		(*-----------------------Weiterschaltbedingungen----------------------------*)
		IF gb_memEndOfBandMarkNIO THEN
			fb_state_entry.i16_next_step := 370;
		ELSE
			IF gst_datensatz.st_md.b_tagreader_fahrend THEN
				(* Pille sofort beschreiben *)
				fb_state_entry.i16_next_step := 350;
			ELSE
				IF st_drive_cmd.enu_cmd = NO_COMMAND THEN
					(* Warte mit Pille beschreiben, bis der Bestücktisch im Ziel ist *)
					fb_state_entry.i16_next_step := 350;
				END_IF
			END_IF
		END_IF


		IF	gst_datensatz.st_md.b_wt_transport_aktiv =FALSE THEN
			visu.b_merker_vollbestuecken:= FALSE;
			s_alte_artikelnummer := '';
			fb_state_entry.i16_next_step := 360;
		END_IF

		IF fb_state_entry.X THEN
			Teile_nach_Bandwechsel:= FALSE;
			IF gst_datensatz.st_wkz.i16_anzahl_Teile_autostop_bandwechsel <> 0 THEN
				gi16_anzahl_Teile_autostop_bandwechsel := gi16_anzahl_Teile_autostop_bandwechsel + 1;
			END_IF
		END_IF

(*=======================================================*)
	350: (* Schreibe Daten auf Tag *)
		IF fb_state_entry.E THEN
			(* Auswertung der Bestückung (Pins bzw. Rasterplatte) des ISK *)
			ST_Markiere_WT_IO();
		END_IF

		(*-----------------------Weiterschaltbedingungen----------------------------*)
		IF balluff_tag_reader.st_ctrl.out.b_fertig AND NOT fb_state_entry.E THEN
			balluff_tag_reader.st_ctrl.in.b_start_schreiben := FALSE;
			fb_state_entry.i16_next_step := 360;
		END_IF

(*=======================================================*)
	360:	(* Aktualisiere letztes benutzes Werkzeug *)
		IF fb_state_entry.E THEN
			ST_Schreibe_LastUsedTool();
		END_IF

		(*-----------------------Weiterschaltbedingungen----------------------------*)
		IF balluff_tag_reader.st_ctrl.out.b_fertig AND NOT fb_state_entry.E THEN
			balluff_tag_reader.st_ctrl.in.b_start_schreiben := FALSE;
			IF gst_datensatz.st_md.b_tagreader_fahrend THEN
				fb_state_entry.i16_next_step := 370;
			ELSE
				fb_state_entry.i16_next_step := 380;
				fb_Z_Achse_ausfahren(b_start:= FALSE, t_zeit=>t_Z_Achse_ausfahren );
			END_IF
		END_IF

(*=======================================================*)
	370:	(* Warte noch auf die Z-Achse, bis sie auf der Übergabeposition steht. *)

		gb_memEndOfBandMarkNIO := FALSE;

		(*-----------------------Weiterschaltbedingungen----------------------------*)
		IF st_drive_cmd.enu_cmd = NO_COMMAND THEN
			fb_state_entry.i16_next_step := 380;
			fb_Z_Achse_ausfahren(b_start:= FALSE, t_zeit=>t_Z_Achse_ausfahren );
		END_IF

(*=======================================================*)
	380:

		CASE gst_datensatz.st_md.i16_typ_zelle OF
			KEINE_ZELLE:
				;

			BESTUECKZELLE_1700:
				(*-----------------------Weiterschaltbedingungen----------------------------*)
				fb_state_entry.i16_next_step := BEREIT;

			RASTERFOLIE:
				(*-----------------------Weiterschaltbedingungen----------------------------*)
				IF rasterfolienmontage.st_ctrl.out.b_fertig_2 THEN
					fb_state_entry.i16_next_step := BEREIT;
				END_IF
		END_CASE

		IF fb_state_entry.X THEN
			(* Stoppe Bestückzeit *)
			zeit_wt_bestuecken := TIME_TO_DWORD(fb_ton_taktzeitmessung_bestuecken.ET);
			fb_ton_taktzeitmessung_bestuecken.IN := FALSE;
			(* Starte WT Wechselzeit *)
			fb_ton_taktzeitmessung_wt_wechsel.IN := TRUE;
		END_IF

(*==========================Bestückzelle1720=============================*)
	395: (*Warten bis keine ander Produktions Meldung ansteht *)
		IF	TestAndSet(ST_Message_Produktion.LockFlag) THEN
			ST_Message_Produktion.ClearMessageLines();
			fb_state_entry.i16_next_step := 396;
		END_IF

(*=======================================================*)
	396:  (*Produktions Meldung*)
		Visu.MeldungProduktion.Color_R := 255;
		Visu.MeldungProduktion.Color_G := 0;
		Visu.MeldungProduktion.Color_B := 0;
		IF visu.s_akt_sprache = 'de' THEN
			Visu.MeldungProduktion.Name:='Zelle war nicht in Betrieb, bitte Instandhalter informieren!$R$N$R$NÖler,Bestückposition, Seitenversatz und Biegewinkel kontrollieren$R$NMeldung kann nur eingeloggt quittiert werden';
		ELSIF visu.s_akt_sprache = 'en' THEN
			Visu.MeldungProduktion.Name:='Station has not been used for last order, please inform Maintenance Technician!$R$N$R$Ncheck oiler, stich position, left/right and bending angle$R$Nmessage can only be acknowledged when logged in';
		ELSIF visu.s_akt_sprache = 'cz' THEN
			Visu.MeldungProduktion.Name:='Bunka nebyla v provozu, informujte prosim serizovace. Zkontrolujte olej, nastaveni os a uhel ohybu.$R$NZprávu lze potvrdit jen po prihlaseni ';
		END_IF
		Visu.MeldungProduktion.ShowMessage := TRUE;
		Visu.MeldungProduktion.Button1.sichtbar:=TRUE;	(*OK*)
		Visu.MeldungProduktion.Button1.Text:='Ok';

		(*-----------------------Weiterschaltbedingungen----------------------------*)
		IF visu.b_logon THEN
			IF Visu.MeldungProduktion.Button1.tasten THEN
				IF gst_datensatz.st_md.	b_tagreader_fahrend THEN
					fb_state_entry.i16_next_step := 400;
				ELSE
					fb_state_entry.i16_next_step := 405;
				END_IF
			END_IF
		END_IF

		IF fb_state_entry.X THEN
			gst_PersDaten.b_Zelle_nicht_in_Betrieb := FALSE;
		END_IF

(*=======================================================*)
	400:	(* Fahre Z-Achse bis auf die erste Bestückposition *)
		IF fb_state_entry.E THEN
			(* Z-Achse verfahren *)
			fb_axis.lr_soll_geschwindigkeit := gst_datensatz.st_wkz.r_auto_z;
			fb_axis.st_position.r_soll := gst_datensatz.st_isk.lr_pos_z_0 + gst_datensatz.st_wkz.lr_offset_z_pos_0 + gst_datensatz.st_wt.lr_offset_z_pos_0 + gst_datensatz.st_md.lr_offset_z_pos_0 + gst_datensatz.st_bestueckprogramm.lr_z[0];
			st_drive_cmd.enu_cmd := MOVE_ABSOLUTE;
		END_IF

		(*-----------------------Weiterschaltbedingungen----------------------------*)
		(* Z-Achse losfahren und währenddessen beschreibt der Tagreader die Pille *)
		fb_state_entry.i16_next_step := 405;

(*=======================================================*)
	405:	(*  WT als schlecht markieren*)
		IF fb_state_entry.E THEN
			ST_Markiere_WT_NIO();
		END_IF

		(*-----------------------Weiterschaltbedingungen----------------------------*)
		IF balluff_tag_reader.st_ctrl.out.b_fertig AND NOT fb_state_entry.E THEN
			(* Ok: Daten sind auf der Pille *)
			balluff_tag_reader.st_ctrl.in.b_start_schreiben := FALSE;
			IF gst_datensatz.st_md.b_tagreader_fahrend THEN
				(* Warte auf Z-Achse *)
				fb_state_entry.i16_next_step := 410;
			ELSE
				(* Daten geschrieben und erst jetzt die Z-Achse fahren *)
				fb_state_entry.i16_next_step := 420;
			END_IF
		END_IF

(*=======================================================*)
	410:	(* Warte noch auf die Z-Achse, bis sie im Ziel steht. *)

		(*-----------------------Weiterschaltbedingungen----------------------------*)
		IF st_drive_cmd.enu_cmd = NO_COMMAND THEN
			fb_state_entry.i16_next_step := 430;
		END_IF

(*=======================================================*)
	420:	(* Fahre Z-Achse bis auf die erste Bestückposition *)
		IF fb_state_entry.E THEN
			(* Z-Achse verfahren *)
			fb_axis.lr_soll_geschwindigkeit := gst_datensatz.st_wkz.r_auto_z;
			fb_axis.st_position.r_soll := gst_datensatz.st_isk.lr_pos_z_0 + gst_datensatz.st_wkz.lr_offset_z_pos_0 + gst_datensatz.st_wt.lr_offset_z_pos_0 + gst_datensatz.st_md.lr_offset_z_pos_0 + gst_datensatz.st_bestueckprogramm.lr_z[0];
			st_drive_cmd.enu_cmd := MOVE_ABSOLUTE;
		END_IF

		(*-----------------------Weiterschaltbedingungen----------------------------*)
		IF st_drive_cmd.enu_cmd = NO_COMMAND THEN
			fb_state_entry.i16_next_step := 430;
		END_IF

(*=======================================================*)
	430:	(* Führung wird an die Bestückachse abgegeben und die Z-Achse wird ausschliesslich über Kurvenscheiben-Kopplung verfahren *)
		IF fb_state_entry.E THEN
			fb_Z_Achse_einfahren(b_start:= FALSE, t_zeit=> t_Z_Achse_einfahren);
			fb_Bestueckung(b_start:= TRUE, t_zeit=> );
			axis_virt_master.st_ctrl.in.b_start := TRUE;

			(* Stoppe WT Wechselzeit *)
			zeit_wt_wechsel := TIME_TO_DWORD(fb_ton_taktzeitmessung_wt_wechsel.ET);
			fb_ton_taktzeitmessung_wt_wechsel.IN := FALSE;

			(* Starte Bestückzeit *)
			fb_ton_taktzeitmessung_bestuecken.IN := TRUE;
		END_IF

		(*-----------------------Weiterschaltbedingungen----------------------------*)
		IF NOT axis_virt_master.st_ctrl.out.b_fertig THEN
			axis_virt_master.st_ctrl.in.b_start := FALSE;
			fb_state_entry.i16_next_step := 440;
		END_IF

		IF fb_state_entry.X THEN
			(* Stoppe Bestückzeit *)
			zeit_wt_bestuecken := TIME_TO_DWORD(fb_ton_taktzeitmessung_bestuecken.ET);
			fb_ton_taktzeitmessung_bestuecken.IN := FALSE;

			(* Starte WT Wechselzeit *)
			fb_ton_taktzeitmessung_wt_wechsel.IN := TRUE;
		END_IF

(*=======================================================*)
	440:	(* Warte auf  Bestückachse fertig mit Pins setzen *)

		(*-----------------------Weiterschaltbedingungen----------------------------*)
		IF axis_virt_master.st_ctrl.out.b_fertig THEN
			fb_state_entry.i16_next_step := 450;
			fb_Bestueckung(b_start:=FALSE, t_zeit=>t_Bestueckung);
			fb_Z_Achse_ausfahren(b_start:= TRUE, t_zeit=> );
		END_IF

(*=======================================================*)
	450: (* Fahre Z-Achse zurück zur Übergabeposition *)
		IF fb_state_entry.E THEN
			 fb_axis.st_position.r_soll := gst_datensatz.st_md.st_md_z_achse.lr_wt_uebergabepos;
			st_drive_cmd.enu_cmd := MOVE_ABSOLUTE;
		END_IF

		(*Nach einem Bandwechsel soll nach X-Teilen gestoppt werden.*)
		IF gst_datensatz.st_wkz.i16_anzahl_Teile_autostop_bandwechsel > 0 THEN
			IF gi16_anzahl_Teile_autostop_bandwechsel = gst_datensatz.st_wkz.i16_anzahl_Teile_autostop_bandwechsel THEN
				gb_nach_bawe_einzelfertigung := TRUE;
			END_IF
		END_IF

		(*-----------------------Weiterschaltbedingungen----------------------------*)
		IF gst_datensatz.st_md.b_tagreader_fahrend THEN
			(* Pille sofort beschreiben *)
			fb_state_entry.i16_next_step := 460;
		ELSE
			IF st_drive_cmd.enu_cmd = NO_COMMAND THEN
				(* Warte mit Pille beschreiben *)
				fb_state_entry.i16_next_step := 460;
			END_IF
		END_IF

		IF	gst_datensatz.st_md.b_wt_transport_aktiv =FALSE THEN
			visu.b_merker_vollbestuecken:= FALSE;
			s_alte_artikelnummer := '';
			fb_state_entry.i16_next_step := 480;
		END_IF

		IF fb_state_entry.X THEN
			IF gst_datensatz.st_wkz.i16_anzahl_Teile_autostop_bandwechsel <> 0 THEN
				gi16_anzahl_Teile_autostop_bandwechsel := gi16_anzahl_Teile_autostop_bandwechsel + 1;
			END_IF
		END_IF

(*=======================================================*)
	460: (* Schreibe Daten auf Tag *)
		IF fb_state_entry.E THEN
			(* WT Hat die Maschine auf regulärem Weg wieder verlassen *)
			ST_Markiere_WT_IO();
		END_IF

		(*-----------------------Weiterschaltbedingungen----------------------------*)
		IF balluff_tag_reader.st_ctrl.out.b_fertig AND NOT fb_state_entry.E THEN
			balluff_tag_reader.st_ctrl.in.b_start_schreiben := FALSE;
			fb_state_entry.i16_next_step := 470;
		END_IF

(*=======================================================*)
	470:	(* aktualisiere letztes benutzes Werkzeug *)
		IF fb_state_entry.E THEN
			ST_Schreibe_LastUsedTool();
		END_IF

		IF balluff_tag_reader.st_ctrl.out.b_fertig AND NOT fb_state_entry.E THEN
			balluff_tag_reader.st_ctrl.in.b_start_schreiben := FALSE;
			IF gst_datensatz.st_md.b_tagreader_fahrend THEN
				fb_state_entry.i16_next_step := 480;
			ELSE
				fb_Z_Achse_ausfahren(b_start:= FALSE, t_zeit=> );
				fb_state_entry.i16_next_step := BEREIT;
			END_IF
		END_IF

(*=======================================================*)
	480:	(* Z-Achse ist fertig positioniert *)

		(*-----------------------Weiterschaltbedingungen----------------------------*)
		IF st_drive_cmd.enu_cmd = NO_COMMAND THEN
			fb_Z_Achse_ausfahren(b_start:= FALSE, t_zeit=> );
			fb_state_entry.i16_next_step := BEREIT;
		END_IF

(*=======================================================*)
	FEHLER:
		IF fb_state_entry.E THEN
			st_ctrl_out.b_fehler := TRUE;
			fb_ton_quitt.IN := FALSE;
			st_ctrl_out.b_busy:=FALSE;
		END_IF

		(*-----------------------Weiterschaltbedingungen----------------------------*)
		IF st_ctrl_in.b_quitt AND NOT fb_state_entry.E THEN
			st_ctrl_out.b_fehler := FALSE;
			st_drive_cmd.enu_cmd := RESET;
			st_drive_cmd_y_achse.enu_cmd := RESET;
			fb_ton_quitt.IN := TRUE;
		END_IF

		IF st_ctrl_in.b_stop AND NOT z_achse.Status.HasBeenStopped THEN
			st_drive_cmd.enu_cmd := STOP_AXIS;
		END_IF

		IF st_ctrl_in.b_halt AND z_achse.Status.Moving THEN
			st_drive_cmd.enu_cmd := HALT_AXIS;
			st_geschwindigkeiten.lr_verzoegerung := lr_decceleration_nothalt;
		END_IF

		IF fb_ton_quitt.Q THEN
			fb_ton_quitt.IN := FALSE;
			fb_state_entry.i16_next_step := INIT;
		END_IF

(*=======================================================*)
	STOP:
		IF fb_state_entry.E THEN
			st_ctrl_out.b_busy:=FALSE;
			IF z_achse.NcToPlc.CoupleState = 0 THEN
				st_drive_cmd.enu_cmd := STOP_AXIS;
			END_IF
		END_IF

		(*-----------------------Weiterschaltbedingungen----------------------------*)
		IF st_drive_cmd.enu_cmd = NO_COMMAND AND z_achse.Status.NotMoving THEN
			fb_state_entry.i16_next_step := STILLSTAND;
		END_IF

(*=======================================================*)
	STILLSTAND:
		IF fb_state_entry.E THEN
			st_drive_cmd.enu_cmd := POWER_DISABLE;
			fb_ton_quitt.IN := FALSE;
		END_IF

		(*-----------------------Weiterschaltbedingungen----------------------------*)
		IF st_ctrl_in.b_quitt AND NOT fb_state_entry.E THEN
			fb_ton_quitt.IN := TRUE;
		END_IF

		IF fb_ton_quitt.Q THEN
			fb_ton_quitt.IN := FALSE;
			fb_state_entry.i16_next_step := INIT;
		END_IF

(*=======================================================*)
	HALT:
		IF fb_state_entry.E THEN
			IF z_achse.NcToPlc.CoupleState = 0 THEN
				st_drive_cmd.enu_cmd := HALT_AXIS;
				st_geschwindigkeiten.lr_verzoegerung := lr_decceleration_nothalt;
			END_IF
			fb_ton_quitt.IN := FALSE;
		END_IF

		(*-----------------------Weiterschaltbedingungen----------------------------*)
		IF st_ctrl_in.b_quitt AND NOT fb_state_entry.E THEN
			fb_ton_quitt.IN := TRUE;
		END_IF

		IF fb_ton_quitt.Q THEN
			fb_ton_quitt.IN := FALSE;
			fb_state_entry.i16_next_step := INIT;
		END_IF

(*=======================================================*)
	HANDRAD:	(* Überprüfe Nullpunktverschiebung des Absolutwertgebers auf Korrektheit *)
		IF fb_state_entry.E THEN
			st_ctrl_out.b_fehler := TRUE;
			fb_axis.i16_nc_parameter_nummer := AxisEncoderOffset;
			st_drive_cmd.enu_cmd := READ_NC_PARAMETER;
		END_IF

		(*-----------------------Weiterschaltbedingungen----------------------------*)
		IF st_drive_cmd.enu_cmd = NO_COMMAND THEN
			IF fb_axis.r_wert_nc_read_parameter = gst_datensatz.st_md.st_md_z_achse.lr_nullpunktverschiebung THEN
				fb_state_entry.i16_next_step := 2040;	(* Jogbetrieb *)
			ELSE
				fb_state_entry.i16_next_step := 2010;	(* Reglerfreigabe nehmen und Nullpunktverschiebung schreiben *)
			END_IF
		END_IF

(*=======================================================*)
	2010:	(* Reglerfreigabe wegnehmen , damit Nullpunktverschiebung geschrieben werden kannt*)
		IF fb_state_entry.E THEN
			st_drive_cmd.enu_cmd := POWER_DISABLE;
		END_IF

		(*-----------------------Weiterschaltbedingungen----------------------------*)
		IF st_drive_cmd.enu_cmd = NO_COMMAND THEN
			fb_state_entry.i16_next_step := 2020;
		END_IF

(*=======================================================*)
	2020:	(* Nullpunktverschiebung hat sich geändert, deshalb erst Null reinschreiben, um keinen Additionsfehler zu machen, *)
			(* weil der Wert der Verschiebung beim Neustart komplett auf die Achse geschrieben wird *)
		IF fb_state_entry.E THEN
			fb_axis.i16_nc_parameter_nummer := AxisEncoderOffset;
			fb_axis.r_wert_nc_write_parameter := 0.0;
			st_drive_cmd.enu_cmd := WRITE_NC_PARAMETER;
		END_IF

		(*-----------------------Weiterschaltbedingungen----------------------------*)
		IF st_drive_cmd.enu_cmd = NO_COMMAND THEN
			fb_state_entry.i16_next_step := 2030;
		END_IF

(*=======================================================*)
	2030:	(* Aktuelle Nullpunktverschiebung des Absolutwertgebers an die Achse senden *)
		IF fb_state_entry.E THEN
			fb_axis.i16_nc_parameter_nummer := AxisEncoderOffset;
			fb_axis.r_wert_nc_write_parameter := gst_datensatz.st_md.st_md_z_achse.lr_nullpunktverschiebung;
			st_drive_cmd.enu_cmd := WRITE_NC_PARAMETER;
		END_IF

		(*-----------------------Weiterschaltbedingungen----------------------------*)
		IF st_drive_cmd.enu_cmd = NO_COMMAND THEN
			fb_state_entry.i16_next_step := 2040;
		END_IF

(*=======================================================*)
	2040:	(* Jogbetrieb *)
		IF fb_state_entry.E THEN
			fb_axis.lr_soll_geschwindigkeit := st_geschwindigkeiten.lr_jog;
		END_IF

		IF ST_Euchner_Handbedienpult.i16_Handrad_delta > 0 THEN
			st_drive_cmd.enu_cmd := JOG_VORWAERTS;
		ELSIF ST_Euchner_Handbedienpult.i16_Handrad_delta < 0 THEN
			st_drive_cmd.enu_cmd := JOG_RUECKWAERTS;
		ELSE
			IF z_achse.Status.Moving THEN
				st_drive_cmd.enu_cmd := JOG_STOP;
			END_IF
		END_IF

		(*-----------------------Weiterschaltbedingungen----------------------------*)
		IF gi16_betriebsart <> HAND OR NOT b_hand_dialog_aktiv THEN
			fb_state_entry.i16_next_step := 2050;
		END_IF

(*=======================================================*)
	2050:
		IF fb_state_entry.E THEN
			st_drive_cmd.enu_cmd := ABORT;
		END_IF

		(*-----------------------Weiterschaltbedingungen----------------------------*)
		IF st_drive_cmd.enu_cmd = NO_COMMAND THEN
			fb_state_entry.i16_next_step := 2060;
		END_IF

(*=======================================================*)
	2060:	(* Reglerfreigabe wegnehmen *)
		IF fb_state_entry.E THEN
			st_drive_cmd.enu_cmd := POWER_DISABLE;
		END_IF

		(*-----------------------Weiterschaltbedingungen----------------------------*)
		IF st_drive_cmd.enu_cmd = NO_COMMAND THEN
			st_ctrl_out.b_fehler := FALSE;
			fb_state_entry.i16_next_step := INIT;
		END_IF

(*=======================================================*)
	NULLPUNKT_SETZEN:
		(* Aktuellen Jog beenden, sonst Probleme beim Softwareendschalter*)
		IF fb_state_entry.E THEN
			st_drive_cmd.enu_cmd := JOG_STOP;
		END_IF

		(*-----------------------Weiterschaltbedingungen----------------------------*)
		IF st_drive_cmd.enu_cmd = NO_COMMAND THEN
			fb_state_entry.i16_next_step := 2505;
		END_IF

(*=======================================================*)
	2505:
		(* 	Lese aktuelle Nullpunkt verschiebung von der Hardware. Der Benutze könnte einen falschen
			Wert eingetragen haben *)
		IF fb_state_entry.E THEN
			fb_axis.i16_nc_parameter_nummer := AxisEncoderOffset;
			st_drive_cmd.enu_cmd := READ_NC_PARAMETER;
		END_IF

		(*-----------------------Weiterschaltbedingungen----------------------------*)
		IF st_drive_cmd.enu_cmd = NO_COMMAND THEN
			gst_datensatz.st_md.st_md_z_achse.lr_nullpunktverschiebung := fb_axis.r_wert_nc_read_parameter;
			fb_state_entry.i16_next_step := 2510;
		END_IF

(*=======================================================*)
	2510:	(* Nullpunktverschiebung berechnen *)
		IF fb_state_entry.E THEN
			lr_pos_ohneverschiebung := axis_z_achse.st_visu.lr_position_ist - gst_datensatz.st_md.st_md_z_achse.lr_nullpunktverschiebung;

			gst_datensatz.st_md.st_md_z_achse.lr_nullpunktverschiebung := - lr_pos_ohneverschiebung;
		END_IF

		(*-----------------------Weiterschaltbedingungen----------------------------*)
		(* Aktiviere den Wert in die Hardware *)
		fb_state_entry.i16_next_step := HANDRAD;

(*=======================================================*)
	INBETRIEBNAHME:	(* Überprüfe Nullpunktverschiebung des Absolutwertgebers auf Korrektheit *)
		IF fb_state_entry.E THEN
			fb_axis.i16_nc_parameter_nummer := AxisEncoderOffset;
			st_drive_cmd.enu_cmd := READ_NC_PARAMETER;
		END_IF

		(*-----------------------Weiterschaltbedingungen----------------------------*)
		IF st_drive_cmd.enu_cmd = NO_COMMAND THEN
			IF fb_axis.r_wert_nc_read_parameter = gst_datensatz.st_md.st_md_z_achse.lr_nullpunktverschiebung THEN
				fb_state_entry.i16_next_step := 5100;	(* Reversiersequenz*)
			ELSE
				fb_state_entry.i16_next_step := 5010;	(* Reglerfreigabe nehmen und Nullpunktverschiebung schreiben *)
			END_IF
		END_IF

(*=======================================================*)
	5010:	(* Reglerfreigabe wegnehmen, damit Nullpunktverschiebung geschrieben werden kannt*)
		IF fb_state_entry.E THEN
			st_drive_cmd.enu_cmd := POWER_DISABLE;
		END_IF

		(*-----------------------Weiterschaltbedingungen----------------------------*)
		IF st_drive_cmd.enu_cmd = NO_COMMAND THEN
			fb_state_entry.i16_next_step := 5020;
		END_IF

(*=======================================================*)
	5020:	(* Nullpunktverschiebung hat sich geändert, deshalb erst Null reinschreiben, um keinen Additionsfehler zu machen, *)
			(* weil der Wert der Verschiebung beim Neustart komplett auf die Achse geschrieben wird *)
		IF fb_state_entry.E THEN
			fb_axis.i16_nc_parameter_nummer := AxisEncoderOffset;
			fb_axis.r_wert_nc_write_parameter := 0.0;
			st_drive_cmd.enu_cmd := WRITE_NC_PARAMETER;
		END_IF

		(*-----------------------Weiterschaltbedingungen----------------------------*)
		IF st_drive_cmd.enu_cmd = NO_COMMAND THEN
			fb_state_entry.i16_next_step := 5030;
		END_IF

(*=======================================================*)
	5030:	(* Aktuelle Nullpunktverschiebung des Absolutwertgebers an die Achse senden *)
		IF fb_state_entry.E THEN
			fb_axis.i16_nc_parameter_nummer := AxisEncoderOffset;
			fb_axis.r_wert_nc_write_parameter := gst_datensatz.st_md.st_md_z_achse.lr_nullpunktverschiebung;
			st_drive_cmd.enu_cmd := WRITE_NC_PARAMETER;
		END_IF

		(*-----------------------Weiterschaltbedingungen----------------------------*)
		IF st_drive_cmd.enu_cmd = NO_COMMAND THEN
			fb_state_entry.i16_next_step := 5100;
		END_IF

(*=======================================================*)
	5100:	(* Verfahren der Achse zwischen zwei Punkten zum Testen verschiedener Achsparameter *)
		IF fb_state_entry.E THEN
			fb_axis.lr_soll_geschwindigkeit := st_geschwindigkeiten.lr_jog;
			fb_axis.st_position.lr_ibn_pos_start := 10.0;
			fb_axis.st_position.lr_ibn_pos_ziel := -10.0;
		END_IF

		(*-----------------------Weiterschaltbedingungen----------------------------*)
		IF st_ctrl_in.b_ibn_start THEN
			fb_state_entry.i16_next_step := 5110;
		END_IF

(*=======================================================*)
	5110: (* Fahre Z-Achse auf Startposition *)
(*
		IF fb_state_entry.E THEN
			 fb_axis.st_position.r_soll := fb_axis.st_position.lr_ibn_pos_start;
			st_drive_cmd.enu_cmd := MOVE_ABSOLUTE;
		END_IF

		(*-----------------------Weiterschaltbedingungen----------------------------*)
		IF st_drive_cmd.enu_cmd = NO_COMMAND THEN
			fb_state_entry.i16_next_step := 5120;
		END_IF
*)
		IF fb_state_entry.E THEN
			st_drive_cmd.enu_cmd := POWER_ENABLE;
		END_IF

		(*-----------------------Weiterschaltbedingungen----------------------------*)
		IF st_drive_cmd.enu_cmd = NO_COMMAND THEN
			;
		END_IF

(*=======================================================*)
	5120: (* Pause *)
		IF fb_state_entry.E THEN
			fb_ton_wz.PT := t#500ms;
			fb_ton_wz.IN := TRUE;
		END_IF

		(*-----------------------Weiterschaltbedingungen----------------------------*)
		IF fb_ton_wz.Q THEN
			fb_ton_wz.IN := FALSE;
			fb_state_entry.i16_next_step := 5130;
		END_IF

(*=======================================================*)
	5130: (* Fahre Z-Achse auf Zielposition *)
		IF fb_state_entry.E THEN
			 fb_axis.st_position.r_soll := fb_axis.st_position.lr_ibn_pos_ziel;
			st_drive_cmd.enu_cmd := MOVE_ABSOLUTE;
		END_IF

		(*-----------------------Weiterschaltbedingungen----------------------------*)
		IF st_drive_cmd.enu_cmd = NO_COMMAND THEN
			fb_state_entry.i16_next_step := 5140;
		END_IF

(*=======================================================*)
	5140: (* Pause *)
		IF fb_state_entry.E THEN
			fb_ton_wz.PT := t#500ms;
			fb_ton_wz.IN := TRUE;
		END_IF

		(*-----------------------Weiterschaltbedingungen----------------------------*)
		IF fb_ton_wz.Q THEN
			fb_ton_wz.IN := FALSE;
			fb_state_entry.i16_next_step := 5100;
		END_IF
END_CASE

fb_state_entry(
	i16_next_step:= ,
	i16_pos:= 2,
	s_debugtext:= ,
	E=> ,
	X=> ,
	i16_step=> ,
	i16_last_step=> );

IF st_config_achse.b_config_fertig THEN
	(* Fehlermeldungen und Betriebsmeldungen ab dem Startindex in die globalen Meldungsarrays schreiben *)
	garr_stoermeldungen[st_config_achse.i16_meld_startindex + 0] := st_sm.b_achse_nicht_bb;
	garr_stoermeldungen[st_config_achse.i16_meld_startindex + 1] := st_sm.b_achse_nicht_referenziert;
	garr_stoermeldungen[st_config_achse.i16_meld_startindex + 2] := st_sm.b_keine_verfahrfreigabe;
	garr_stoermeldungen[st_config_achse.i16_meld_startindex + 3] := st_sm.b_achse_nicht_auf_startpos;
	garr_stoermeldungen[st_config_achse.i16_meld_startindex + 4] := st_sm.b_ende_skalierungs_nocke;
	garr_stoermeldungen[st_config_achse.i16_meld_startindex + 5] := st_sm.b_ende_camming_nocke;
	garr_stoermeldungen[st_config_achse.i16_meld_startindex + 6] := st_sm.b_skalierung_noch_aktiv;
	garr_stoermeldungen[st_config_achse.i16_meld_startindex + 7] := FALSE;
	garr_stoermeldungen[st_config_achse.i16_meld_startindex + 8] := FALSE;
	garr_stoermeldungen[st_config_achse.i16_meld_startindex + 9] := FALSE;
	garr_stoermeldungen[st_config_achse.i16_meld_startindex + 10] := sm_positionsueberwachung;
	garr_stoermeldungen[st_config_achse.i16_meld_startindex + 11] := sm_werkzeugreihenfolge_nicht_io;
	garr_stoermeldungen[st_config_achse.i16_meld_startindex + 12] := sm_keine_bandfreigabe;
	garr_stoermeldungen[st_config_achse.i16_meld_startindex + 13] := sm_tagnummer_ungueltig;
	garr_stoermeldungen[st_config_achse.i16_meld_startindex + 14] := FALSE;
	garr_stoermeldungen[st_config_achse.i16_meld_startindex + 15] := sm_typ_bestueckprogramm_falsch;
	garr_stoermeldungen[st_config_achse.i16_meld_startindex + 16] := st_drive_cmd.meldungen.sm_write_soe_parameter;
	garr_stoermeldungen[st_config_achse.i16_meld_startindex + 17] := st_drive_cmd.meldungen.sm_read_soe_parameter;
	garr_stoermeldungen[st_config_achse.i16_meld_startindex + 18] := st_drive_cmd.meldungen.sm_write_nc_parameter;
	garr_stoermeldungen[st_config_achse.i16_meld_startindex + 19] := st_drive_cmd.meldungen.sm_read_nc_parameter;
	garr_stoermeldungen[st_config_achse.i16_meld_startindex + 20] := st_drive_cmd.meldungen.sm_power_enable;
	garr_stoermeldungen[st_config_achse.i16_meld_startindex + 21] := st_drive_cmd.meldungen.sm_power_disable;
	garr_stoermeldungen[st_config_achse.i16_meld_startindex + 22] := st_drive_cmd.meldungen.sm_reset;
	garr_stoermeldungen[st_config_achse.i16_meld_startindex + 23] := st_drive_cmd.meldungen.sm_home;
	garr_stoermeldungen[st_config_achse.i16_meld_startindex + 24] := st_drive_cmd.meldungen.sm_setposition;
	garr_stoermeldungen[st_config_achse.i16_meld_startindex + 25] := st_drive_cmd.meldungen.sm_jog_vorwaerts;
	garr_stoermeldungen[st_config_achse.i16_meld_startindex + 26] := st_drive_cmd.meldungen.sm_jog_rueckwaerts;
	garr_stoermeldungen[st_config_achse.i16_meld_startindex + 27] := st_drive_cmd.meldungen.sm_move_absolute;
	garr_stoermeldungen[st_config_achse.i16_meld_startindex + 28] := st_drive_cmd.meldungen.sm_move_relative;
	garr_stoermeldungen[st_config_achse.i16_meld_startindex + 29] := st_drive_cmd.meldungen.sm_move_velocity;
	garr_stoermeldungen[st_config_achse.i16_meld_startindex + 30] := st_drive_cmd.meldungen.sm_move_modulo;
	garr_stoermeldungen[st_config_achse.i16_meld_startindex + 31] := st_drive_cmd.meldungen.sm_stop_axis;
	garr_stoermeldungen[st_config_achse.i16_meld_startindex + 32] := st_drive_cmd.meldungen.sm_halt_axis;
	garr_stoermeldungen[st_config_achse.i16_meld_startindex + 33] := st_drive_cmd.meldungen.sm_motion_command_timeout;
	garr_stoermeldungen[st_config_achse.i16_meld_startindex + 34] := st_sm.b_achsfehler;
	garr_stoermeldungen[st_config_achse.i16_meld_startindex + 35] := st_sm.b_devicefehler;
	garr_stoermeldungen[st_config_achse.i16_meld_startindex + 36] := st_drive_cmd.meldungen.sm_limit_positiv_erreicht;
	garr_stoermeldungen[st_config_achse.i16_meld_startindex + 37] := st_drive_cmd.meldungen.sm_limit_negativ_erreicht;
	garr_stoermeldungen[st_config_achse.i16_meld_startindex + 38] := st_drive_cmd.meldungen.sm_ec_coe_sdo_write_ex;
	garr_stoermeldungen[st_config_achse.i16_meld_startindex + 39] := st_drive_cmd.meldungen.sm_ec_coe_sdo_read_ex;
	garr_stoermeldungen[st_config_achse.i16_meld_startindex + 40] := st_drive_cmd_y_achse.meldungen.sm_gear_in_slave;
	garr_stoermeldungen[st_config_achse.i16_meld_startindex + 41] := st_drive_cmd_y_achse.meldungen.sm_gear_out_slave;
	garr_stoermeldungen[st_config_achse.i16_meld_startindex + 42] := st_drive_cmd_y_achse.meldungen.sm_cam_in_slave;
	garr_stoermeldungen[st_config_achse.i16_meld_startindex + 43] := st_drive_cmd_y_achse.meldungen.sm_cam_out_slave;
	garr_stoermeldungen[st_config_achse.i16_meld_startindex + 44] := st_drive_cmd_y_achse.meldungen.sm_cam_scaleing_slave;
	garr_stoermeldungen[st_config_achse.i16_meld_startindex + 45] := st_drive_cmd_y_achse.meldungen.sm_camgear_command_timeout;;
	garr_stoermeldungen[st_config_achse.i16_meld_startindex + 46] := st_drive_cmd_y_achse.meldungen.sm_read_motion_funktion_point;
	garr_stoermeldungen[st_config_achse.i16_meld_startindex + 47] := st_drive_cmd_y_achse.meldungen.sm_write_motion_funktion_point;
	garr_stoermeldungen[st_config_achse.i16_meld_startindex + 48] := st_drive_cmd_y_achse.meldungen.sm_read_camtable_slave_dynamics;
	garr_stoermeldungen[st_config_achse.i16_meld_startindex + 49] := st_drive_cmd_y_achse.meldungen.sm_read_camtable_charakteristik;
	garr_stoermeldungen[st_config_achse.i16_meld_startindex + 50] := FALSE;
	garr_stoermeldungen[st_config_achse.i16_meld_startindex + 51] := FALSE;
	garr_stoermeldungen[st_config_achse.i16_meld_startindex + 52] := FALSE;
	garr_stoermeldungen[st_config_achse.i16_meld_startindex + 53] := FALSE;
	garr_stoermeldungen[st_config_achse.i16_meld_startindex + 54] := FALSE;
	garr_stoermeldungen[st_config_achse.i16_meld_startindex + 55] := FALSE;
	garr_stoermeldungen[st_config_achse.i16_meld_startindex + 56] := FALSE;
	garr_stoermeldungen[st_config_achse.i16_meld_startindex + 57] := FALSE;
	garr_stoermeldungen[st_config_achse.i16_meld_startindex + 58] := FALSE;
	garr_stoermeldungen[st_config_achse.i16_meld_startindex + 59] := FALSE;
	garr_stoermeldungen[st_config_achse.i16_meld_startindex + 60] := FALSE;
	garr_stoermeldungen[st_config_achse.i16_meld_startindex + 61] := FALSE;
	garr_stoermeldungen[st_config_achse.i16_meld_startindex + 62] := FALSE;
	garr_stoermeldungen[st_config_achse.i16_meld_startindex + 63] := FALSE;
	garr_stoermeldungen[st_config_achse.i16_meld_startindex + 64] := FALSE;
	garr_stoermeldungen[st_config_achse.i16_meld_startindex + 65] := FALSE;
	garr_stoermeldungen[st_config_achse.i16_meld_startindex + 66] := FALSE;
	garr_stoermeldungen[st_config_achse.i16_meld_startindex + 67] := FALSE;
	garr_stoermeldungen[st_config_achse.i16_meld_startindex + 68] := FALSE;
	garr_stoermeldungen[st_config_achse.i16_meld_startindex + 69] := FALSE;
	garr_stoermeldungen[st_config_achse.i16_meld_startindex + 70] := FALSE;
	garr_stoermeldungen[st_config_achse.i16_meld_startindex + 71] := FALSE;
	garr_stoermeldungen[st_config_achse.i16_meld_startindex + 72] := FALSE;
	garr_stoermeldungen[st_config_achse.i16_meld_startindex + 73] := FALSE;
	garr_stoermeldungen[st_config_achse.i16_meld_startindex + 74] := FALSE;
	garr_stoermeldungen[st_config_achse.i16_meld_startindex + 75] := FALSE;
	garr_stoermeldungen[st_config_achse.i16_meld_startindex + 76] := FALSE;
	garr_stoermeldungen[st_config_achse.i16_meld_startindex + 77] := FALSE;
	garr_stoermeldungen[st_config_achse.i16_meld_startindex + 78] := FALSE;
	garr_stoermeldungen[st_config_achse.i16_meld_startindex + 79] := FALSE;
	garr_stoermeldungen[st_config_achse.i16_meld_startindex + 80] := FALSE;
	garr_stoermeldungen[st_config_achse.i16_meld_startindex + 81] := FALSE;
	garr_stoermeldungen[st_config_achse.i16_meld_startindex + 82] := FALSE;
	garr_stoermeldungen[st_config_achse.i16_meld_startindex + 83] := FALSE;
	garr_stoermeldungen[st_config_achse.i16_meld_startindex + 84] := FALSE;
	garr_stoermeldungen[st_config_achse.i16_meld_startindex + 85] := FALSE;
	garr_stoermeldungen[st_config_achse.i16_meld_startindex + 86] := FALSE;
	garr_stoermeldungen[st_config_achse.i16_meld_startindex + 87] := FALSE;
	garr_stoermeldungen[st_config_achse.i16_meld_startindex + 88] := FALSE;
	garr_stoermeldungen[st_config_achse.i16_meld_startindex + 89] := FALSE;
	garr_stoermeldungen[st_config_achse.i16_meld_startindex + 90] := FALSE;
	garr_stoermeldungen[st_config_achse.i16_meld_startindex + 91] := FALSE;
	garr_stoermeldungen[st_config_achse.i16_meld_startindex + 92] := FALSE;
	garr_stoermeldungen[st_config_achse.i16_meld_startindex + 93] := FALSE;
	garr_stoermeldungen[st_config_achse.i16_meld_startindex + 94] := FALSE;
	garr_stoermeldungen[st_config_achse.i16_meld_startindex + 95] := FALSE;
	garr_stoermeldungen[st_config_achse.i16_meld_startindex + 96] := FALSE;
	garr_stoermeldungen[st_config_achse.i16_meld_startindex + 97] := FALSE;
	garr_stoermeldungen[st_config_achse.i16_meld_startindex + 98] := FALSE;
	garr_stoermeldungen[st_config_achse.i16_meld_startindex + 99] := FALSE;
	
	garr_betriebsmeldungen[st_config_achse.i16_meld_startindex + 0] := bm_kein_Pin_im_BB;
	garr_betriebsmeldungen[st_config_achse.i16_meld_startindex + 1] := bm_rastnasen_1_fehlt;
	garr_betriebsmeldungen[st_config_achse.i16_meld_startindex + 2] := bm_rastnasen_2_fehlt;
	garr_betriebsmeldungen[st_config_achse.i16_meld_startindex + 3] := FALSE;
	garr_betriebsmeldungen[st_config_achse.i16_meld_startindex + 4] := FALSE;
	garr_betriebsmeldungen[st_config_achse.i16_meld_startindex + 5] := FALSE;
	garr_betriebsmeldungen[st_config_achse.i16_meld_startindex + 6] := FALSE;
	garr_betriebsmeldungen[st_config_achse.i16_meld_startindex + 7] := FALSE;
	garr_betriebsmeldungen[st_config_achse.i16_meld_startindex + 8] := FALSE;
	garr_betriebsmeldungen[st_config_achse.i16_meld_startindex + 9] := FALSE;
	garr_betriebsmeldungen[st_config_achse.i16_meld_startindex + 10] := FALSE;
	garr_betriebsmeldungen[st_config_achse.i16_meld_startindex + 11] := FALSE;
	garr_betriebsmeldungen[st_config_achse.i16_meld_startindex + 12] := FALSE;
	garr_betriebsmeldungen[st_config_achse.i16_meld_startindex + 13] := FALSE;
	garr_betriebsmeldungen[st_config_achse.i16_meld_startindex + 14] := FALSE;
	garr_betriebsmeldungen[st_config_achse.i16_meld_startindex + 15] := FALSE;
	garr_betriebsmeldungen[st_config_achse.i16_meld_startindex + 16] := FALSE;
	garr_betriebsmeldungen[st_config_achse.i16_meld_startindex + 17] := FALSE;
	garr_betriebsmeldungen[st_config_achse.i16_meld_startindex + 18] := FALSE;
	garr_betriebsmeldungen[st_config_achse.i16_meld_startindex + 19] := FALSE;
	garr_betriebsmeldungen[st_config_achse.i16_meld_startindex + 20] := FALSE;
	garr_betriebsmeldungen[st_config_achse.i16_meld_startindex + 21] := FALSE;
	garr_betriebsmeldungen[st_config_achse.i16_meld_startindex + 22] := FALSE;
	garr_betriebsmeldungen[st_config_achse.i16_meld_startindex + 23] := FALSE;
	garr_betriebsmeldungen[st_config_achse.i16_meld_startindex + 24] := FALSE;
	garr_betriebsmeldungen[st_config_achse.i16_meld_startindex + 25] := FALSE;
	garr_betriebsmeldungen[st_config_achse.i16_meld_startindex + 26] := FALSE;
	garr_betriebsmeldungen[st_config_achse.i16_meld_startindex + 27] := FALSE;
	garr_betriebsmeldungen[st_config_achse.i16_meld_startindex + 28] := FALSE;
	garr_betriebsmeldungen[st_config_achse.i16_meld_startindex + 29] := FALSE;
	garr_betriebsmeldungen[st_config_achse.i16_meld_startindex + 30] := FALSE;
	garr_betriebsmeldungen[st_config_achse.i16_meld_startindex + 31] := FALSE;
	garr_betriebsmeldungen[st_config_achse.i16_meld_startindex + 32] := FALSE;
	garr_betriebsmeldungen[st_config_achse.i16_meld_startindex + 33] := FALSE;
	garr_betriebsmeldungen[st_config_achse.i16_meld_startindex + 34] := FALSE;
	garr_betriebsmeldungen[st_config_achse.i16_meld_startindex + 35] := FALSE;
	garr_betriebsmeldungen[st_config_achse.i16_meld_startindex + 36] := FALSE;
	garr_betriebsmeldungen[st_config_achse.i16_meld_startindex + 37] := FALSE;
	garr_betriebsmeldungen[st_config_achse.i16_meld_startindex + 38] := FALSE;
	garr_betriebsmeldungen[st_config_achse.i16_meld_startindex + 39] := FALSE;
	garr_betriebsmeldungen[st_config_achse.i16_meld_startindex + 40] := FALSE;
	garr_betriebsmeldungen[st_config_achse.i16_meld_startindex + 41] := FALSE;
	garr_betriebsmeldungen[st_config_achse.i16_meld_startindex + 42] := FALSE;
	garr_betriebsmeldungen[st_config_achse.i16_meld_startindex + 43] := FALSE;
	garr_betriebsmeldungen[st_config_achse.i16_meld_startindex + 44] := FALSE;
	garr_betriebsmeldungen[st_config_achse.i16_meld_startindex + 45] := FALSE;
	garr_betriebsmeldungen[st_config_achse.i16_meld_startindex + 46] := FALSE;
	garr_betriebsmeldungen[st_config_achse.i16_meld_startindex + 47] := FALSE;
	garr_betriebsmeldungen[st_config_achse.i16_meld_startindex + 48] := FALSE;
	garr_betriebsmeldungen[st_config_achse.i16_meld_startindex + 49] := FALSE;
END_IF
END_PROGRAM

(* POU EPT Lib/Funktionsbausteine/ST_Taktzeit, ST *)
FUNCTION_BLOCK ST_Taktzeit
VAR_INPUT
	b_start			: BOOL;
END_VAR
VAR_OUTPUT
	t_zeit			: TIME;
END_VAR
VAR
	fb_f_trig_stop		: F_TRIG;
	fb_ton			: TON;
END_VAR
fb_f_trig_stop(CLK:= b_start, Q=> );

IF fb_f_trig_stop.Q THEN
	t_zeit := fb_ton.ET;
END_IF

fb_ton(IN:= b_start, PT:= t#20h, Q=> );
END_FUNCTION_BLOCK

(* POU Gemeinsamkeiten17xx/Achsen/ST_MotionFunctionPoints, ST *)
PROGRAM ST_MotionFunctionPoints
VAR_INPUT
	st_ctrl_in								: struct_ctrl_in;
END_VAR
VAR_OUTPUT
	st_ctrl_out							: struct_ctrl_out;
END_VAR
VAR
	fb_ton_wz							: TON;
	fb_ton_quitt							: TON;
	fb_state_entry						: ST_StateEntry;
	i, j									: INT := 0;
	udi_table_id_bestueckachse			: UDINT := 0;
	arr_motion_function_points		: ARRAY[1..ARRAY_LAENGE_MFP] OF struct_db_motionfunctionpoint;
END_VAR
VAR CONSTANT
	ARRAY_LAENGE_MFP				: INT := 100;
	YZTischMasterPos2					 : LREAL := 125;
	YZTischMasterPos3					 : LREAL := 185;
END_VAR
(* Zeiten *)
fb_ton_wz(IN:= ,PT:= , Q=>  , ET=> );
fb_ton_quitt(IN:= , PT:= t#50ms, Q=> , ET=> );

(* =====Berechnung MFPs===== *)
(* Berechnung von Punkten in einer Kurvenscheibe und der maximalen Mastergeschwindigkeit *)

(* =====Kopplung: Virtuelle Masterachse <-> Z-Achse ===== *)
fb_edit_mfps_bestuecken_z.fb(
	st_config:= fb_edit_mfps_bestuecken_z.st_config,
	st_ctrl_in:= fb_edit_mfps_bestuecken_z.st_ctrl.in,
	udiTableId:= 1,
	eMotionFunctionType:= MOTIONFUNCTYPE_POLYNOM5,
	i16_startpunkt_edit_mf_tab:= 2,
	arr_db_mf_tab:= arr_motion_function_points,
	lrVeloMax:= ST_Z_Achse.st_geschwindigkeiten.lr_maximalgeschwindigkeit,
	lrAccMax:= ST_Z_Achse.st_geschwindigkeiten.lr_beschleunigung,
	lrDecMax:= ST_Z_Achse.st_geschwindigkeiten.lr_verzoegerung,
	lrModuloValue:= 360.0,
	st_AxisRefMaster:= virtuelle_master_achse,
	st_AxisRefSlave:= z_achse,
	lrMasterVeloMax=> ,		(* Maximum Master Velocity [°/s] *)
	lrMasterRotPerMinMax=> ,	(* Maximum Master Rotations per Minute [1/min] *)
	st_ctrl_out=> fb_edit_mfps_bestuecken_z.st_ctrl.out);

(* =====Kopplung: Virtuelle Masterachse <-> Y-Achse ===== *)
fb_edit_mfps_bestuecken_y.fb(
	st_config:= fb_edit_mfps_bestuecken_y.st_config,
	st_ctrl_in:= fb_edit_mfps_bestuecken_y.st_ctrl.in,
	udiTableId:= 3,
	eMotionFunctionType:= MOTIONFUNCTYPE_POLYNOM5,
	i16_startpunkt_edit_mf_tab:= 2,
	arr_db_mf_tab:= arr_motion_function_points,
	lrVeloMax:= ST_Y_Achse.st_geschwindigkeiten.lr_maximalgeschwindigkeit,
	lrAccMax:= ST_Y_Achse.st_geschwindigkeiten.lr_beschleunigung,
	lrDecMax:= ST_Y_Achse.st_geschwindigkeiten.lr_verzoegerung,
	lrModuloValue:= 360.0,
	st_AxisRefMaster:= virtuelle_master_achse,
	st_AxisRefSlave:= y_achse,
	lrMasterVeloMax=> ,		(* Maximum Master Velocity [°/s] *)
	lrMasterRotPerMinMax=> ,	(* Maximum Master Rotations per Minute [1/min] *)
	st_ctrl_out=> fb_edit_mfps_bestuecken_y.st_ctrl.out);

(* =====Kopplung: Virtuelle Masterachse <-> Servobandeinzug-Achse ===== *)
fb_edit_mfps_bestuecken_b.fb(
	st_config:= fb_edit_mfps_bestuecken_b.st_config,
	st_ctrl_in:= fb_edit_mfps_bestuecken_b.st_ctrl.in,
	udiTableId:= 4,
	eMotionFunctionType:= MOTIONFUNCTYPE_POLYNOM5,
	i16_startpunkt_edit_mf_tab:= 2,
	arr_db_mf_tab:= arr_motion_function_points,
	lrVeloMax:= ST_Servobandeinzug.st_geschwindigkeiten.lr_maximalgeschwindigkeit,
	lrAccMax:= ST_Servobandeinzug.st_geschwindigkeiten.lr_beschleunigung,
	lrDecMax:= ST_Servobandeinzug.st_geschwindigkeiten.lr_verzoegerung,
	lrModuloValue:= 360.0,
	st_AxisRefMaster:= bestueckachse,
	st_AxisRefSlave:= b_achse,
	lrMasterVeloMax=> ,		(* Maximum Master Velocity [°/s] *)
	lrMasterRotPerMinMax=> ,	(* Maximum Master Rotations per Minute [1/min] *)
	st_ctrl_out=> fb_edit_mfps_bestuecken_b.st_ctrl.out);

(* =====Kopplung: Z-Achse <-> Y-Achse ===== *)
fb_edit_mfps_yz_tisch.fb(
	st_config:= fb_edit_mfps_yz_tisch.st_config,
	st_ctrl_in:= fb_edit_mfps_yz_tisch.st_ctrl.in,
	udiTableId:= 2,
	eMotionFunctionType:= MOTIONFUNCTYPE_POLYNOM5,
	i16_startpunkt_edit_mf_tab:= 2,
	arr_db_mf_tab:= arr_motion_function_points,
	lrVeloMax:= ST_Y_Achse.st_geschwindigkeiten.lr_maximalgeschwindigkeit,
	lrAccMax:= ST_Y_Achse.st_geschwindigkeiten.lr_beschleunigung,
	lrDecMax:= ST_Y_Achse.st_geschwindigkeiten.lr_verzoegerung,
	lrModuloValue:= 0.0,
	st_AxisRefMaster:= z_achse,
	st_AxisRefSlave:= y_achse,
	lrMasterVeloMax=> ,		(* Maximum Master Velocity [mm/s] *)
	lrMasterRotPerMinMax=> ,	(* Maximum Master Rotations per Minute [1/min] *)
	st_ctrl_out=> fb_edit_mfps_yz_tisch.st_ctrl.out);

(* =====Kopplung: Virtuelle Masterachse <-> Bestueckachse ===== *)
(*
fb_edit_mfps_bestueckachse.fb(
	st_config:= fb_edit_mfps_bestueckachse.st_config,
	st_ctrl_in:= fb_edit_mfps_bestueckachse.st_ctrl.in,
	udiTableId:= udi_table_id_bestueckachse,
	eMotionFunctionType:= MOTIONFUNCTYPE_POLYNOM5,
	i16_startpunkt_edit_mf_tab:= 1,
	arr_db_mf_tab:= gst_datensatz.st_wkz.st_virtmaster_bestueckachse.arr_motion_function_points,
	lrVeloMax:= ST_Bestueckachse.st_geschwindigkeiten.lr_maximalgeschwindigkeit,
	lrAccMax:= ST_Bestueckachse.st_geschwindigkeiten.lr_beschleunigung,
	lrDecMax:= ST_Bestueckachse.st_geschwindigkeiten.lr_verzoegerung,
	lrModuloValue:= 360.0,
	st_AxisRefMaster:= virtuelle_master_achse,
	st_AxisRefSlave:= bestueckachse,
	lrMasterVeloMax=> ,		(* Maximum Master Velocity [°/s] *)
	lrMasterRotPerMinMax=> ,	(* Maximum Master Rotations per Minute [1/min] *)
	st_ctrl_out=> fb_edit_mfps_bestueckachse.st_ctrl.out);
*)
fb_camtable_bestueckachse.fb(
	st_config:= fb_camtable_bestueckachse.st_config,
	st_ctrl_in:= fb_camtable_bestueckachse.st_ctrl.in,
	udiTableId:= udi_table_id_bestueckachse,
	arr_db_mf_tab:= arr_motion_function_points,
	lrModuloValue:= 360,
	st_AxisRefMaster:= virtuelle_master_achse,
	st_AxisRefSlave:= bestueckachse,
	st_ctrl_out=> fb_camtable_bestueckachse.st_ctrl.out);

(* =======================================Toplevel========================================== *)
IF fb_state_entry.i16_next_step > INIT AND fb_state_entry.i16_next_step < FEHLER THEN
	(* =====Fehler MFP-Berechnung===== *)
	IF 	fb_edit_mfps_bestuecken_z.st_ctrl.out.b_fehler OR
		fb_edit_mfps_bestuecken_y.st_ctrl.out.b_fehler OR
		fb_edit_mfps_bestuecken_b.st_ctrl.out.b_fehler OR
		fb_edit_mfps_yz_tisch.st_ctrl.out.b_fehler OR
		fb_camtable_bestueckachse.st_ctrl.out.b_fehler
		THEN
			fb_state_entry.i16_next_step := FEHLER;
	END_IF

	IF fb_state_entry.i16_next_step < STOP THEN
		IF st_ctrl_in.b_stop THEN
			fb_state_entry.i16_next_step := STOP;
		END_IF
	END_IF
END_IF

(* ======================================Schrittkette======================================== *)
fb_state_entry(
	i16_next_step:= ,
	i16_pos:= 1,
	s_debugtext:= ,
	E=> ,
	X=> ,
	i16_step=> ,
	i16_last_step=> );

CASE fb_state_entry.i16_step OF
	INIT_OBJ:
		fb_state_entry.i16_next_step := INIT;

(*=======================================================*)
	INIT:
		IF fb_state_entry.E THEN
			fb_ton_wz.IN := FALSE;
			fb_ton_quitt.IN := FALSE;
			st_ctrl_out.b_fehler := FALSE;
			st_ctrl_out.b_fertig := FALSE;
			st_ctrl_out.b_bereit := FALSE;

			fb_edit_mfps_bestuecken_z.st_ctrl.in.b_start := FALSE;
			fb_edit_mfps_bestuecken_y.st_ctrl.in.b_start := FALSE;
			fb_edit_mfps_bestuecken_b.st_ctrl.in.b_start := FALSE;
			fb_edit_mfps_yz_tisch.st_ctrl.in.b_start := FALSE;
			fb_camtable_bestueckachse.st_ctrl.in.b_start := FALSE;
		END_IF

		(*-----------------------Weiterschaltbedingungen----------------------------*)
		IF st_ctrl_in.b_init THEN
			fb_edit_mfps_bestuecken_z.st_ctrl.in.b_quitt := FALSE;
			fb_edit_mfps_bestuecken_y.st_ctrl.in.b_quitt := FALSE;
			fb_edit_mfps_bestuecken_b.st_ctrl.in.b_quitt := FALSE;
			fb_edit_mfps_yz_tisch.st_ctrl.in.b_quitt := FALSE;
			fb_camtable_bestueckachse.st_ctrl.in.b_quitt := FALSE;

			CASE gst_datensatz.st_md.i16_typ_zelle OF
				KEINE_ZELLE:
					;

				BESTUECKZELLE_1700:
					fb_state_entry.i16_next_step := 20;

				BESTUECKZELLE_1720:
					fb_state_entry.i16_next_step := 40;

				RASTERFOLIE:
					fb_state_entry.i16_next_step := 50;
			END_CASE
		END_IF

(*===========================MFP berechnen============================*)
	20:	(* Initialisierung der Kurvenscheibenwerte für Bestückachse-ZAchse aus der DB -> grundlegende Definition der Motionfunktion *)
		(* 1700 *)
		IF fb_state_entry.E THEN
			(* Kurvenscheibe Best-Z-Achse *)
			subr_ST_MFP_Z_Achse();
		END_IF

		(*-----------------------Weiterschaltbedingungen----------------------------*)
		IF fb_edit_mfps_bestuecken_z.fb.st_ctrl_out.b_fertig AND NOT fb_state_entry.E THEN
			fb_edit_mfps_bestuecken_z.st_ctrl.in.b_start := FALSE;
			fb_state_entry.i16_next_step := 21;
		END_IF

(*=======================================================*)
	21:	(* 1700 *)
		IF fb_state_entry.E THEN
			(* Kurvenscheibe Best-Y-Achse *)
			subr_ST_MFP_Y_Achse();
		END_IF

		(*-----------------------Weiterschaltbedingungen----------------------------*)
		IF fb_edit_mfps_bestuecken_y.fb.st_ctrl_out.b_fertig AND NOT fb_state_entry.E THEN
			fb_edit_mfps_bestuecken_y.st_ctrl.in.b_start := FALSE;
			fb_state_entry.i16_next_step := 22;
		END_IF

(*=======================================================*)
	22:	(* 1700 *)
		IF fb_state_entry.E THEN
			(* Kurvenscheibe Y-Z-Tisch *)
			subr_ST_MFP_YZ_Tisch();
		END_IF

		(*-----------------------Weiterschaltbedingungen----------------------------*)
		IF fb_edit_mfps_yz_tisch.st_ctrl.out.b_fertig AND NOT fb_state_entry.E THEN
			fb_edit_mfps_yz_tisch.st_ctrl.in.b_start := FALSE;
			fb_state_entry.i16_next_step := 23;
		END_IF

(*=======================================================*)
	23:	(* 1700 *)
		IF fb_state_entry.E THEN
			(* Kurvenscheibe mit Scalierung 1 Virtuelle Masterachse - Bestückachse *)
			subr_ST_MFP_Bestueckachse_S1();
		END_IF

		(*-----------------------Weiterschaltbedingungen----------------------------*)
		IF fb_camtable_bestueckachse.st_ctrl.out.b_fertig AND NOT fb_state_entry.E THEN
			fb_camtable_bestueckachse.st_ctrl.in.b_start := FALSE;
			fb_state_entry.i16_next_step := 24;
		END_IF

(*=======================================================*)
	24:	(* 1700 *)
		IF fb_state_entry.E THEN
			(* Kurvenscheibe mit Scalierung 0 Virtuelle Masterachse - Bestückachse *)
			subr_ST_MFP_Bestueckachse_S0();
		END_IF

		(*-----------------------Weiterschaltbedingungen----------------------------*)
		IF fb_camtable_bestueckachse.st_ctrl.out.b_fertig AND NOT fb_state_entry.E THEN
			fb_camtable_bestueckachse.st_ctrl.in.b_start := FALSE;
			fb_state_entry.i16_next_step := 25;
		END_IF

(*=======================================================*)
	25:	(* 1700 *)
		IF fb_state_entry.E THEN
			CASE gst_datensatz.st_wkz.i16_typ_bandeinzug OF
				BANDWECHSLER_V2:
					fb_state_entry.i16_next_step := BEREIT;
				SERVO:
					(* Kurvenscheibe Best-Servobandeinzug-Achse *)
					subr_ST_MFP_B_Achse();
			END_CASE;
		END_IF

		(*-----------------------Weiterschaltbedingungen----------------------------*)
		IF fb_edit_mfps_bestuecken_b.fb.st_ctrl_out.b_fertig AND NOT fb_state_entry.E THEN
			fb_edit_mfps_bestuecken_b.st_ctrl.in.b_start := FALSE;
			fb_state_entry.i16_next_step := BEREIT;
		END_IF

(*=======================================================*)
	30:	(* Initialisierung der Kurvenscheibenwerte für Bestückachse-ZAchse aus der DB -> grundlegende Definition der Motionfunktion *)
		(* RASTERPLATTE *)
		IF fb_state_entry.E THEN
			(* Kurvenscheibe Y-Z-Tisch *)
			subr_ST_MFP_YZ_Tisch();
		END_IF

		(*-----------------------Weiterschaltbedingungen----------------------------*)
		IF fb_edit_mfps_yz_tisch.st_ctrl.out.b_fertig AND NOT fb_state_entry.E THEN
			fb_edit_mfps_yz_tisch.st_ctrl.in.b_start := TRUE;
			fb_state_entry.i16_next_step := BEREIT;
		END_IF

(*=======================================================*)
	40:	(* Initialisierung der Kurvenscheibenwerte für Bestückachse-ZAchse aus der DB -> grundlegende Definition der Motionfunktion *)
		(* 1720 *)
		IF fb_state_entry.E THEN
			(* Kurvenscheibe Best-Z-Achse *)
			FOR i := 1 TO ARRAY_LAENGE_MFP BY 1DO
				arr_motion_function_points[i].PointIndex := i;
				arr_motion_function_points[i].FunctionType := MOTIONFUNCTYPE_NOTDEF;
				arr_motion_function_points[i].PointType := MOTIONPOINTTYPE_IGNORE;
				arr_motion_function_points[i].MasterPos := 0.0;
				arr_motion_function_points[i].SlavePos := 0.0;
			END_FOR
			FOR i := 1 TO 4 BY 1DO
				arr_motion_function_points[i].PointIndex := i;
				arr_motion_function_points[i].FunctionType := MOTIONFUNCTYPE_POLYNOM1;
				arr_motion_function_points[i].PointType := MOTIONPOINTTYPE_VELOCITY;
			END_FOR
			arr_motion_function_points[2].FunctionType := MOTIONFUNCTYPE_POLYNOM5_MM;
			arr_motion_function_points[1].MasterPos := 0.0;
			arr_motion_function_points[1].SlavePos := 0.0;
			arr_motion_function_points[2].MasterPos := 250;
			arr_motion_function_points[2].SlavePos := 0.0;
			arr_motion_function_points[3].MasterPos := 340;
			arr_motion_function_points[3].SlavePos := 1;
			arr_motion_function_points[4].MasterPos := 360;
			arr_motion_function_points[4].SlavePos := 1;
			fb_edit_mfps_bestuecken_z.st_ctrl.in.b_start := TRUE;
		END_IF

		(*-----------------------Weiterschaltbedingungen----------------------------*)
		IF fb_edit_mfps_bestuecken_z.fb.st_ctrl_out.b_fertig AND NOT fb_state_entry.E THEN
			fb_edit_mfps_bestuecken_z.st_ctrl.in.b_start := FALSE;
			fb_state_entry.i16_next_step := 41;
		END_IF

(*=======================================================*)
	41:	(* 1720 *)
		IF fb_state_entry.E THEN
			(* Kurvenscheibe mit Scalierung 1 Virtuelle Masterachse - Bestückachse *)
			subr_ST_MFP_Bestueckachse_S1();
		END_IF

		(*-----------------------Weiterschaltbedingungen----------------------------*)
		IF fb_camtable_bestueckachse.st_ctrl.out.b_fertig AND NOT fb_state_entry.E THEN
			fb_camtable_bestueckachse.st_ctrl.in.b_start := FALSE;
			fb_state_entry.i16_next_step := 42;
		END_IF

(*=======================================================*)
	42:	(* 1720 *)
		IF fb_state_entry.E THEN
			(* Kurvenscheibe mit Scalierung 0 Virtuelle Masterachse - Bestückachse *)
			subr_ST_MFP_Bestueckachse_S0();
		END_IF

		(*-----------------------Weiterschaltbedingungen----------------------------*)
		IF fb_camtable_bestueckachse.st_ctrl.out.b_fertig AND NOT fb_state_entry.E THEN
			fb_camtable_bestueckachse.st_ctrl.in.b_start := FALSE;
			fb_state_entry.i16_next_step := BEREIT;
		END_IF

(*=======================================================*)
	50:	(* Rasterfolie *)
		IF fb_state_entry.E THEN
			(* Kurvenscheibe Best-Z-Achse *)
			subr_ST_MFP_Z_Achse();
		END_IF

		(*-----------------------Weiterschaltbedingungen----------------------------*)
		IF fb_edit_mfps_bestuecken_z.fb.st_ctrl_out.b_fertig AND NOT fb_state_entry.E THEN
			fb_edit_mfps_bestuecken_z.st_ctrl.in.b_start := FALSE;
			fb_state_entry.i16_next_step := 51;
		END_IF

(*=======================================================*)
	51:	(* Rasterfolie *)
		IF fb_state_entry.E THEN
			(* Kurvenscheibe Best-Y-Achse *)
			subr_ST_MFP_Y_Achse();
		END_IF

		(*-----------------------Weiterschaltbedingungen----------------------------*)
		IF fb_edit_mfps_bestuecken_y.fb.st_ctrl_out.b_fertig AND NOT fb_state_entry.E THEN
			fb_edit_mfps_bestuecken_y.st_ctrl.in.b_start := FALSE;
			fb_state_entry.i16_next_step := 52;
		END_IF

(*=======================================================*)
	52:	(* Rasterfolie *)
		IF fb_state_entry.E THEN
			(* Kurvenscheibe Y-Z-Tisch *)
			FOR i := 1 TO ARRAY_LAENGE_MFP BY 1DO
				arr_motion_function_points[i].PointIndex := i;
				arr_motion_function_points[i].FunctionType := MOTIONFUNCTYPE_NOTDEF;
				arr_motion_function_points[i].PointType := MOTIONPOINTTYPE_IGNORE;
				arr_motion_function_points[i].MasterPos := 0.0;
				arr_motion_function_points[i].SlavePos := 0.0;
			END_FOR
			FOR i := 1 TO 4 BY 1DO
				arr_motion_function_points[i].PointIndex := i;
				arr_motion_function_points[i].FunctionType := MOTIONFUNCTYPE_POLYNOM1;
				arr_motion_function_points[i].PointType := MOTIONPOINTTYPE_VELOCITY;
			END_FOR
			arr_motion_function_points[2].FunctionType := MOTIONFUNCTYPE_POLYNOM5_MM;
			arr_motion_function_points[1].MasterPos := -115;
			arr_motion_function_points[1].SlavePos := gst_datensatz.st_wkz.st_yz_tisch.r_wkz_einfahrpos_y;
			arr_motion_function_points[2].MasterPos := gst_datensatz.st_wkz.st_yz_tisch.r_wkz_einfahrpos_z;
			arr_motion_function_points[2].SlavePos := gst_datensatz.st_wkz.st_yz_tisch.r_wkz_einfahrpos_y;
			arr_motion_function_points[3].MasterPos := 175;
			arr_motion_function_points[3].SlavePos := gst_datensatz.st_md.st_md_y_achse.lr_wt_uebergabepos;
			arr_motion_function_points[4].MasterPos := 200;
			arr_motion_function_points[4].SlavePos := gst_datensatz.st_md.st_md_y_achse.lr_wt_uebergabepos;
			fb_edit_mfps_yz_tisch.st_ctrl.in.b_start := TRUE;
		END_IF

		(*-----------------------Weiterschaltbedingungen----------------------------*)
		IF fb_edit_mfps_yz_tisch.st_ctrl.out.b_fertig AND NOT fb_state_entry.E THEN
			fb_edit_mfps_yz_tisch.st_ctrl.in.b_start := FALSE;
			fb_state_entry.i16_next_step := 53;
		END_IF

(*=======================================================*)
	53:	(* Rasterfolie *)
		IF fb_state_entry.E THEN
			(* Kurvenscheibe mit Scalierung 1 Virtuelle Masterachse - Bestückachse *)
			subr_ST_MFP_Bestueckachse_S1();
		END_IF

		(*-----------------------Weiterschaltbedingungen----------------------------*)
		IF fb_camtable_bestueckachse.st_ctrl.out.b_fertig AND NOT fb_state_entry.E THEN
			fb_camtable_bestueckachse.st_ctrl.in.b_start := FALSE;
			fb_state_entry.i16_next_step := 54;
		END_IF

(*=======================================================*)
	54:	(* Rasterfolie *)
		IF fb_state_entry.E THEN
			(* Kurvenscheibe mit Scalierung 0 Virtuelle Masterachse - Bestückachse *)
			subr_ST_MFP_Bestueckachse_S0();
		END_IF

		(*-----------------------Weiterschaltbedingungen----------------------------*)
		IF fb_camtable_bestueckachse.st_ctrl.out.b_fertig AND NOT fb_state_entry.E THEN
			fb_camtable_bestueckachse.st_ctrl.in.b_start := FALSE;
			fb_state_entry.i16_next_step := BEREIT;
		END_IF

(*=======================================================*)
	BEREIT:
		IF fb_state_entry.E THEN
			st_ctrl_out.b_bereit := TRUE;
		END_IF

(*=======================================================*)
	FEHLER:
		IF fb_state_entry.E THEN
			st_ctrl_out.b_fehler := TRUE;
			fb_ton_quitt.IN := FALSE;
			fb_edit_mfps_bestuecken_z.st_ctrl.in.b_quitt := FALSE;
			fb_edit_mfps_bestuecken_y.st_ctrl.in.b_quitt := FALSE;
			fb_edit_mfps_bestuecken_b.st_ctrl.in.b_quitt := FALSE;
			fb_edit_mfps_yz_tisch.st_ctrl.in.b_quitt := FALSE;
			fb_camtable_bestueckachse.st_ctrl.in.b_quitt := FALSE;
		END_IF

		(*-----------------------Weiterschaltbedingungen----------------------------*)
		IF st_ctrl_in.b_quitt AND NOT fb_state_entry.E THEN
			st_ctrl_out.b_fehler := FALSE;
			fb_ton_quitt.IN := TRUE;
			fb_edit_mfps_bestuecken_z.st_ctrl.in.b_quitt := TRUE;
			fb_edit_mfps_bestuecken_y.st_ctrl.in.b_quitt := TRUE;
			fb_edit_mfps_bestuecken_b.st_ctrl.in.b_quitt := TRUE;
			fb_edit_mfps_yz_tisch.st_ctrl.in.b_quitt := TRUE;
			fb_camtable_bestueckachse.st_ctrl.in.b_quitt := TRUE;
		END_IF

		IF fb_ton_quitt.Q THEN
			fb_ton_quitt.IN := FALSE;
			fb_state_entry.i16_next_step := INIT;
		END_IF

(*=======================================================*)
	STOP:
		IF fb_state_entry.E THEN
			fb_ton_quitt.IN := FALSE;
			fb_edit_mfps_bestuecken_z.st_ctrl.in.b_quitt := FALSE;
			fb_edit_mfps_bestuecken_y.st_ctrl.in.b_quitt := FALSE;
			fb_edit_mfps_bestuecken_b.st_ctrl.in.b_quitt := FALSE;
			fb_edit_mfps_yz_tisch.st_ctrl.in.b_quitt := FALSE;
			fb_camtable_bestueckachse.st_ctrl.in.b_quitt := FALSE;
		END_IF

		(*-----------------------Weiterschaltbedingungen----------------------------*)
		IF st_ctrl_in.b_quitt AND NOT fb_state_entry.E THEN
			fb_ton_quitt.IN := TRUE;
			fb_edit_mfps_bestuecken_z.st_ctrl.in.b_quitt := TRUE;
			fb_edit_mfps_bestuecken_y.st_ctrl.in.b_quitt := TRUE;
			fb_edit_mfps_bestuecken_b.st_ctrl.in.b_quitt := TRUE;
			fb_edit_mfps_yz_tisch.st_ctrl.in.b_quitt := TRUE;
			fb_camtable_bestueckachse.st_ctrl.in.b_quitt := TRUE;
		END_IF

		IF fb_ton_quitt.Q THEN
			fb_ton_quitt.IN := FALSE;
			fb_state_entry.i16_next_step := INIT;
		END_IF
END_CASE

fb_state_entry(
	i16_next_step:= , 
	i16_pos:= 2,
	s_debugtext:= ,
	E=> , 
	X=> , 
	i16_step=> ,
	i16_last_step=> );
END_PROGRAM
ACTION subr_ST_MFP_B_Achse:
(* Kurvenscheibe Best-Servobandeinzug-Achse *)
FOR i := 1 TO ARRAY_LAENGE_MFP BY 1DO
	arr_motion_function_points[i].PointIndex := i;
	arr_motion_function_points[i].FunctionType := MOTIONFUNCTYPE_NOTDEF;
	arr_motion_function_points[i].PointType := MOTIONPOINTTYPE_IGNORE;
	arr_motion_function_points[i].MasterPos := 0.0;
	arr_motion_function_points[i].SlavePos := 0.0;
END_FOR
FOR i := 1 TO 5 BY 1DO
	arr_motion_function_points[i].PointIndex := i;
	arr_motion_function_points[i].FunctionType := MOTIONFUNCTYPE_POLYNOM1;
	arr_motion_function_points[i].PointType := MOTIONPOINTTYPE_VELOCITY;
END_FOR
arr_motion_function_points[2].FunctionType := MOTIONFUNCTYPE_POLYNOM5_MM;
arr_motion_function_points[1].MasterPos := 0.0;
arr_motion_function_points[1].SlavePos := 0.0;
arr_motion_function_points[2].MasterPos := 50;
arr_motion_function_points[2].SlavePos := 0.0;
arr_motion_function_points[3].MasterPos := 100;
arr_motion_function_points[3].SlavePos := 1;
arr_motion_function_points[4].MasterPos := 200;
arr_motion_function_points[4].SlavePos := 1;
arr_motion_function_points[5].MasterPos := 360;
arr_motion_function_points[5].SlavePos := 1;
fb_edit_mfps_bestuecken_b.st_ctrl.in.b_start := TRUE;
END_ACTION
ACTION subr_ST_MFP_Bestueckachse_S0:
(* Kurvenscheibe mit Scalierung 0 Virtuelle Masterachse - Bestückachse *)
udi_table_id_bestueckachse := 6;
FOR i := 1 TO ARRAY_LAENGE_MFP BY 1DO
	arr_motion_function_points[i].PointIndex := i;
	arr_motion_function_points[i].FunctionType := MOTIONFUNCTYPE_NOTDEF;
	arr_motion_function_points[i].PointType := MOTIONPOINTTYPE_IGNORE;
	arr_motion_function_points[i].MasterPos := 0.0;
	arr_motion_function_points[i].SlavePos := 0.0;
END_FOR
FOR i := 1 TO 2 BY 1DO
	arr_motion_function_points[i].PointIndex := i;
	arr_motion_function_points[i].FunctionType := MOTIONFUNCTYPE_POLYNOM1;
	arr_motion_function_points[i].PointType := MOTIONPOINTTYPE_VELOCITY;
END_FOR
arr_motion_function_points[1].MasterPos := 0;
arr_motion_function_points[1].SlavePos := gst_datensatz.st_md.st_md_bestueckachse.lr_startposition;
arr_motion_function_points[2].MasterPos := 360;
arr_motion_function_points[2].SlavePos := gst_datensatz.st_md.st_md_bestueckachse.lr_startposition;
fb_camtable_bestueckachse.st_ctrl.in.b_start := TRUE;
END_ACTION
ACTION subr_ST_MFP_Bestueckachse_S1:
(* Kurvenscheibe mit Scalierung 1 Virtuelle Masterachse - Bestückachse *)
udi_table_id_bestueckachse := 5;
FOR i := 1 TO ARRAY_LAENGE_MFP BY 1DO
	arr_motion_function_points[i].PointIndex := i;
	arr_motion_function_points[i].FunctionType := MOTIONFUNCTYPE_NOTDEF;
	arr_motion_function_points[i].PointType := MOTIONPOINTTYPE_IGNORE;
	arr_motion_function_points[i].MasterPos := 0.0;
	arr_motion_function_points[i].SlavePos := 0.0;
END_FOR
FOR i := 1 TO 2 BY 1DO
	arr_motion_function_points[i].PointIndex := i;
	arr_motion_function_points[i].FunctionType := MOTIONFUNCTYPE_POLYNOM1;
	arr_motion_function_points[i].PointType := MOTIONPOINTTYPE_VELOCITY;
END_FOR
arr_motion_function_points[1].MasterPos := 0;
arr_motion_function_points[1].SlavePos := 0;
arr_motion_function_points[2].MasterPos := 360;
arr_motion_function_points[2].SlavePos := 360;
fb_camtable_bestueckachse.st_ctrl.in.b_start := TRUE;
END_ACTION
ACTION subr_ST_MFP_Y_Achse:
(* Kurvenscheibe Best-Y-Achse *)
FOR i := 1 TO ARRAY_LAENGE_MFP BY 1DO
	arr_motion_function_points[i].PointIndex := i;
	arr_motion_function_points[i].FunctionType := MOTIONFUNCTYPE_NOTDEF;
	arr_motion_function_points[i].PointType := MOTIONPOINTTYPE_IGNORE;
	arr_motion_function_points[i].MasterPos := 0.0;
	arr_motion_function_points[i].SlavePos := 0.0;
END_FOR
FOR i := 1 TO 4 BY 1DO
	arr_motion_function_points[i].PointIndex := i;
	arr_motion_function_points[i].FunctionType := MOTIONFUNCTYPE_POLYNOM1;
	arr_motion_function_points[i].PointType := MOTIONPOINTTYPE_VELOCITY;
END_FOR
arr_motion_function_points[2].FunctionType := MOTIONFUNCTYPE_POLYNOM5_MM;
arr_motion_function_points[1].MasterPos := 0.0;
arr_motion_function_points[1].SlavePos := 0.0;
arr_motion_function_points[2].MasterPos := 40;
arr_motion_function_points[2].SlavePos := 0.0;
arr_motion_function_points[3].MasterPos := 260;
arr_motion_function_points[3].SlavePos := 1;
arr_motion_function_points[4].MasterPos := 360;
arr_motion_function_points[4].SlavePos := 1;
fb_edit_mfps_bestuecken_y.st_ctrl.in.b_start := TRUE;
END_ACTION
ACTION subr_ST_MFP_YZ_Tisch:
(* Kurvenscheibe Y-Z-Tisch *)


	CASE gst_datensatz.st_md.i16_typ_zelle OF
			KEINE_ZELLE:
					;

			BESTUECKZELLE_1700, BESTUECKZELLE_1720, RASTERFOLIE:

				FOR i := 1 TO ARRAY_LAENGE_MFP BY 1DO
					arr_motion_function_points[i].PointIndex := i;
					arr_motion_function_points[i].FunctionType := MOTIONFUNCTYPE_NOTDEF;
					arr_motion_function_points[i].PointType := MOTIONPOINTTYPE_IGNORE;
					arr_motion_function_points[i].MasterPos := 0.0;
					arr_motion_function_points[i].SlavePos := 0.0;
				END_FOR
				FOR i := 1 TO 4 BY 1DO
					arr_motion_function_points[i].PointIndex := i;
					arr_motion_function_points[i].FunctionType := MOTIONFUNCTYPE_POLYNOM1;
					arr_motion_function_points[i].PointType := MOTIONPOINTTYPE_VELOCITY;
				END_FOR

				IF gst_datensatz.st_wkz.b_variable_einfahrposition THEN
					arr_motion_function_points[2].FunctionType := MOTIONFUNCTYPE_POLYNOM5_MM;
					arr_motion_function_points[1].MasterPos := -115;
					arr_motion_function_points[1].SlavePos := gst_datensatz.st_wkz.st_yz_tisch.r_wkz_einfahrpos_y;
					arr_motion_function_points[2].MasterPos :=gst_datensatz.st_wkz.st_yz_tisch.r_wkz_einfahrpos_z;
					arr_motion_function_points[2].SlavePos := gst_datensatz.st_wkz.st_yz_tisch.r_wkz_einfahrpos_y;
					arr_motion_function_points[3].MasterPos := YZTischMasterPos3;
					arr_motion_function_points[3].SlavePos := gst_datensatz.st_md.st_md_y_achse.lr_wt_uebergabepos;
					arr_motion_function_points[4].MasterPos := 200;
					arr_motion_function_points[4].SlavePos := gst_datensatz.st_md.st_md_y_achse.lr_wt_uebergabepos;
				ELSE
					arr_motion_function_points[2].FunctionType := MOTIONFUNCTYPE_POLYNOM5_MM;
					arr_motion_function_points[1].MasterPos := -115;
					arr_motion_function_points[1].SlavePos := gst_datensatz.st_wkz.st_yz_tisch.r_wkz_einfahrpos_y;
					arr_motion_function_points[2].MasterPos := YZTischMasterPos2;
					arr_motion_function_points[2].SlavePos := gst_datensatz.st_wkz.st_yz_tisch.r_wkz_einfahrpos_y;
					arr_motion_function_points[3].MasterPos := YZTischMasterPos3;
					arr_motion_function_points[3].SlavePos := gst_datensatz.st_md.st_md_y_achse.lr_wt_uebergabepos;
					arr_motion_function_points[4].MasterPos := 200;
					arr_motion_function_points[4].SlavePos := gst_datensatz.st_md.st_md_y_achse.lr_wt_uebergabepos;
				END_IF
				fb_edit_mfps_yz_tisch.st_ctrl.in.b_start := TRUE;


	END_CASE
END_ACTION
ACTION subr_ST_MFP_Z_Achse:
(* Kurvenscheibe Best-Z-Achse *)
FOR i := 1 TO ARRAY_LAENGE_MFP BY 1DO
	arr_motion_function_points[i].PointIndex := i;
	arr_motion_function_points[i].FunctionType := MOTIONFUNCTYPE_NOTDEF;
	arr_motion_function_points[i].PointType := MOTIONPOINTTYPE_IGNORE;
	arr_motion_function_points[i].MasterPos := 0.0;
	arr_motion_function_points[i].SlavePos := 0.0;
END_FOR
FOR i := 1 TO 4 BY 1DO
	arr_motion_function_points[i].PointIndex := i;
	arr_motion_function_points[i].FunctionType := MOTIONFUNCTYPE_POLYNOM1;
	arr_motion_function_points[i].PointType := MOTIONPOINTTYPE_VELOCITY;
END_FOR
arr_motion_function_points[2].FunctionType := MOTIONFUNCTYPE_POLYNOM5_MM;
arr_motion_function_points[1].MasterPos := 0.0;
arr_motion_function_points[1].SlavePos := 0.0;
arr_motion_function_points[2].MasterPos := 40;
arr_motion_function_points[2].SlavePos := 0.0;
arr_motion_function_points[3].MasterPos := 260;
arr_motion_function_points[3].SlavePos := 1;
arr_motion_function_points[4].MasterPos := 360;
arr_motion_function_points[4].SlavePos := 1;
fb_edit_mfps_bestuecken_z.st_ctrl.in.b_start := TRUE;
END_ACTION

(* POU Gemeinsamkeiten17xx/Achsen/ST_Y_Achse, ST *)
PROGRAM ST_Y_Achse
VAR_INPUT
	st_config_achse						: struct_ecd_config;
	st_ctrl_in								: struct_ctrl_in;
	e_steuerung_ein						: BOOL;
	e_ba_mit_bedingungen				: BOOL;
	e_tuere_vorne_offen					: BOOL;
	e_tuere_hinten_offen					: BOOL;
	e_not_steu_tuer_schutz_ok				: BOOL;
	lr_tmp_Achspos						: LREAL;

	b_start_in							: BOOL;
	lr_Achspos_in						: LREAL;
	lr_Velo_in							: LREAL;
	enu_cmd_in							: enum_ecd_cmd;
END_VAR
VAR_IN_OUT
	st_visu								: struct_ecd_visu;
END_VAR
VAR_OUTPUT
	st_ctrl_out							: struct_ctrl_out;
	lr_RecPos							: LREAL;
END_VAR
VAR
	st_sm						 		: struct_ecd_meldungen;
	st_drive_cmd							: struct_ecd_cmd;
	fb_ton_wz							: TON;
	fb_ton_quitt							: TON;
	fb_ton_wz_disable						: TON;
	fb_r_trig_start							: R_TRIG;
	fb_r_trig_start_in						: R_TRIG;
	fb_r_trig_taste_plus					: R_TRIG;
	fb_r_trig_taste_minus					: R_TRIG;
	fb_r_trig_hand_dialog					: R_TRIG;
	fb_axis								: ST_AxisJobCtrl_Motion;
	fb_state_entry							: ST_StateEntry;
	fb_ton_uez							: TON;
	fb_ton_regelfreigabe_y_achse			: TON;
	i									: UINT := 0;
	lr_pos_ohneverschiebung			: LREAL;
	fb_r_trig_limit_sensor_positiv			: R_TRIG;
	fb_r_trig_limit_sensor_negativ			: R_TRIG;
	fb_r_trig_skalierungsnocken				: R_TRIG;
	fb_r_trig_nullpunkt_setzen				: R_TRIG;

	b_hand_dialog_aktiv					: BOOL := FALSE;
	sm_kein_nocken_definiert				: BOOL := FALSE;

	st_geschwindigkeiten					: struct_ecd_geschwindigkeiten;
	e_referenz_sensor						AT %I* : BOOL;
	i16_torque							AT %I* : INT;
	i16_DigitalInput						AT %I* : INT;

	lr_decceleration_nothalt				: LREAL;
	lr_decceleration_normal				: LREAL;

	i16_state_msg						: INT;
	lr_MaxSoftPosLimit					:LREAL;
	lr_MinSoftPosLimit						:LREAL;
	b_EndlageErreicht						:BOOL;
	fb_r_trig_Endlage						: R_TRIG;
END_VAR
(* Zeiten *)
fb_ton_wz(IN:= , PT:= , Q=>  , ET=> );
fb_ton_uez(IN:= , PT:= , Q=>  , ET=> );
fb_ton_quitt(IN:= , PT:= t#100ms, Q=> , ET=> );
fb_ton_wz_disable(IN:= , PT:= t#500ms, Q=> , ET=> );

(* Flanken *)
fb_r_trig_limit_sensor_positiv(CLK:= st_config_achse.b_limitsensor_positiv_vorhanden AND NOT fb_axis.e_limit_sensor_positive, Q=> );
fb_r_trig_limit_sensor_negativ(CLK:= st_config_achse.b_limitsensor_negativ_vorhanden AND NOT fb_axis.e_limit_sensor_negative, Q=> );
fb_r_trig_taste_plus(CLK:= ST_Euchner_Handbedienpult.b_Taste_Plus, Q=> );
fb_r_trig_taste_minus(CLK:= ST_Euchner_Handbedienpult.b_Taste_Minus, Q=> );
fb_r_trig_start(CLK:= st_ctrl_in.b_start, Q=> );
fb_r_trig_start_in(CLK:= b_start_in, Q=> );
fb_r_trig_skalierungsnocken(CLK:= nockenschaltwerk_bestueckachse.fb.arr_spur[SP_START_SKALIERUNG], Q=> );
fb_r_trig_hand_dialog(CLK:= b_hand_dialog_aktiv, Q=> );
fb_r_trig_nullpunkt_setzen(CLK:=axis_y_achse.st_visu.b_nullpunkt_setzen);

(* Achse steuern *)
fb_axis(
	e_referenznocken:= ,
	b_refsensor_vorhanden:= st_config_achse.b_refsensor_vorhanden,
	b_limitsensor_positiv_vorhanden:= st_config_achse.b_limitsensor_positiv_vorhanden,
	b_limitsensor_negativ_vorhanden:= st_config_achse.b_limitsensor_negativ_vorhanden,
	i16_achstyp := st_config_achse.i16_achstyp,
	lr_override_vorgabe:= ST_TippTasten.lr_override,
	st_position:= ,
	mc_richtung_modulo:= ,
	mc_richtung_velocity:= ,
	mc_referenzmodus:= ,
	mc_buffermode_axis:= ,
	ui16_soeparam_write_value:= ,
	w_idn:= ,
	i16_nc_parameter_nummer:= ,
	r_wert_nc_write_parameter:= ,
	st_vorgabe_geschwindigkeiten:= st_geschwindigkeiten,
	lr_soll_geschwindigkeit:= ,
	b_bedingung_sls:= NOT e_tuere_vorne_offen OR NOT e_tuere_hinten_offen,
	st_ads_info := ,
	st_eccoe_sdo := ,
	st_masterachse:= y_achse,
	st_visu_axis:= st_visu,
	st_ecd_cmd:= st_drive_cmd,
	ui16_soeparam_read_value=> ,
	r_wert_nc_read_parameter=>  ,
	lr_RecPos=> lr_RecPos,
	b_TriggerInput:=i16_DigitalInput.2,
	b_FallingEdge:=TRUE);

(* Achse mit dem Euchner Handbediengerät vorwärts und rückwärts Bewegen*)
IF gi16_betriebsart = HAND AND fb_r_trig_hand_dialog.Q THEN
	fb_state_entry.i16_next_step := HANDRAD;
END_IF

IF gi16_betriebsart = HAND THEN
	(* Button in der Oberfläche zum setzen des Nullpunktes *)
	IF fb_r_trig_nullpunkt_setzen.Q THEN
		fb_state_entry.i16_next_step :=	NULLPUNKT_SETZEN;
	END_IF
END_IF


(*Meldung Achse hat Endlage überfahren*)
IF lr_MinSoftPosLimit<>0 AND
 lr_MinSoftPosLimit > gst_datensatz.st_md.st_md_y_achse.lr_wt_uebergabepos THEN
	b_EndlageErreicht:=TRUE;
ELSE
	b_EndlageErreicht:=FALSE;
END_IF

fb_r_trig_Endlage(CLK:= b_EndlageErreicht , Q=> );

IF fb_r_trig_Endlage.Q THEN
	i16_state_msg := 1;
END_IF

(*Produktionsmeldung für Endlage überfahren*)
CASE i16_state_msg OF
	1: (*Warten bis keine ander Produktions Meldung ansteht *)
		IF	TestAndSet(ST_Message_Produktion.LockFlag) THEN
			ST_Message_Produktion.ClearMessageLines();
			i16_state_msg := 2;
		END_IF

	2:  (*Produktions Meldung*)
		Visu.MeldungProduktion.Color_R := 255;
		Visu.MeldungProduktion.Color_G := 255;
		Visu.MeldungProduktion.Color_B := 0;
		IF visu.s_akt_sprache = 'de' THEN
			Visu.MeldungProduktion.Name:='Y-Achse WT Übergabepos größer als Endlage';
		ELSIF visu.s_akt_sprache = 'en' THEN
			Visu.MeldungProduktion.Name:='Y-Achse WT Übergabepos größer als Endlage';
		ELSIF visu.s_akt_sprache = 'cz' THEN
			Visu.MeldungProduktion.Name:='Y-Achse WT Übergabepos größer als Endlage';
		END_IF
		Visu.MeldungProduktion.ShowMessage := TRUE;
		Visu.MeldungProduktion.Button1.sichtbar:= FALSE;	(*OK*)
		Visu.MeldungProduktion.Button1.Text:='Ok';
		i16_state_msg := 3;

	3:  (*Warte auf OK*)
		IF NOT b_EndlageErreicht THEN
			ST_Message_Produktion.b_PM_Quitt:=TRUE;
			i16_state_msg:=0;
		END_IF
END_CASE

(* =======================================Toplevel========================================== *)
(* Starte Inbetriebnahme-Sequenz *)
IF st_ctrl_in.b_gehe_step_ibn THEN
	fb_state_entry.i16_next_step := INBETRIEBNAHME;
END_IF

(* =====Achse wird disabled===== *)
IF (NOT e_steuerung_ein OR NOT e_ba_mit_bedingungen) AND y_achse.Status.Operational THEN
	st_drive_cmd.enu_cmd := POWER_DISABLE;
END_IF

IF fb_state_entry.i16_next_step > INIT AND fb_state_entry.i16_next_step < FEHLER THEN
	(* =====Fehler vom Achskontroller===== *)
	IF st_drive_cmd.b_job_fehler THEN
		fb_state_entry.i16_next_step := FEHLER;
	END_IF

	IF fb_state_entry.i16_next_step > 35 THEN
		(* Devicefehler *)
		IF y_achse.Status.Error THEN
			st_sm.b_achsfehler := TRUE;
			fb_state_entry.i16_next_step := FEHLER;
		ELSIF y_achse.Status.DriveDeviceError THEN
			st_sm.b_devicefehler := TRUE;
			fb_state_entry.i16_next_step := FEHLER;
		END_IF
	END_IF

	IF fb_state_entry.i16_next_step < STOP THEN
		(* =====Achse wird gestoppt===== *)
		IF st_ctrl_in.b_stop THEN
			fb_state_entry.i16_next_step := STOP;
		ELSIF fb_state_entry.i16_next_step < HALT THEN
			(* =====Achse wird angehalten===== *)
			IF st_ctrl_in.b_halt THEN
				fb_state_entry.i16_next_step := HALT;
			END_IF
		END_IF
	END_IF
END_IF

(* ======================================Schrittkette======================================== *)
fb_state_entry(
	i16_next_step:= ,
	i16_pos:= 1,
	E=> ,
	X=> , 
	i16_step=> ,
	i16_last_step=> );

CASE fb_state_entry.i16_step OF
(*=======================================================*)
	INIT_OBJ:
		IF st_config_achse.b_config_fertig THEN
			fb_state_entry.i16_next_step := 1;
		END_IF

(*=======================================================*)
	1:	(* Warte bis NetID´s der Slaves ausgelesen sind *)
		IF fb_state_entry.E THEN
			;
		END_IF

		(*-----------------------Weiterschaltbedingungen----------------------------*)
		IF ST_EthercatDiag.st_ctrl_out.b_fertig THEN
			fb_state_entry.i16_next_step := 2;
		END_IF

(*=======================================================*)
	2:	(* Spezifische NC-Achsparameter auslesen *)
		IF fb_state_entry.E THEN
			fb_axis.i16_nc_parameter_nummer := MaxVelocitySystem;
			st_drive_cmd.enu_cmd := READ_NC_PARAMETER;
		END_IF

		(*-----------------------Weiterschaltbedingungen----------------------------*)
		IF st_drive_cmd.enu_cmd = NO_COMMAND THEN
			lr_Velo_in:=st_geschwindigkeiten.lr_maximalgeschwindigkeit;
			st_geschwindigkeiten.lr_auto_max := st_geschwindigkeiten.lr_maximalgeschwindigkeit := fb_axis.r_wert_nc_read_parameter;
			st_geschwindigkeiten.lr_auto_min := 25.0;
			st_geschwindigkeiten.lr_jog := 50;
			fb_state_entry.i16_next_step := 3;
		END_IF

(*=======================================================*)
	3:	(* Spezifische NC-Achsparameter auslesen *)
		IF fb_state_entry.E THEN
			fb_axis.i16_nc_parameter_nummer := MaxAccelerationSystem;
			st_drive_cmd.enu_cmd := READ_NC_PARAMETER;
		END_IF

		(*-----------------------Weiterschaltbedingungen----------------------------*)
		IF st_drive_cmd.enu_cmd = NO_COMMAND THEN
			st_geschwindigkeiten.lr_beschleunigung := fb_axis.r_wert_nc_read_parameter;
			fb_state_entry.i16_next_step := 4;
		END_IF

(*=======================================================*)
	4:	(* Spezifische NC-Achsparameter auslesen *)
		IF fb_state_entry.E THEN
			fb_axis.i16_nc_parameter_nummer := MaxDecelerationSystem;
			st_drive_cmd.enu_cmd := READ_NC_PARAMETER;
		END_IF

		(*-----------------------Weiterschaltbedingungen----------------------------*)
		IF st_drive_cmd.enu_cmd = NO_COMMAND THEN
			st_geschwindigkeiten.lr_verzoegerung := fb_axis.r_wert_nc_read_parameter;
			lr_decceleration_normal := st_geschwindigkeiten.lr_verzoegerung;
			lr_decceleration_nothalt := 200000.0;
			fb_state_entry.i16_next_step := 5;
		END_IF

(*=======================================================*)
	5:	(* Spezifische NC-Achsparameter auslesen *)
		IF fb_state_entry.E THEN
			fb_axis.i16_nc_parameter_nummer := MaxJerk;
			st_drive_cmd.enu_cmd := READ_NC_PARAMETER;
		END_IF

		(*-----------------------Weiterschaltbedingungen----------------------------*)
		IF st_drive_cmd.enu_cmd = NO_COMMAND THEN
			st_geschwindigkeiten.lr_ruck := fb_axis.r_wert_nc_read_parameter;
			fb_state_entry.i16_next_step := 6;
		END_IF

(*=======================================================*)
	6:	(* Konfigurationen der Achse *)
		IF fb_state_entry.E THEN
			fb_axis.st_eccoe_sdo.s_ec_slave_net_id := ST_EthercatDiag.s_ec_slave_net_id[2];
			fb_axis.st_eccoe_sdo.ui16_slave_addr := st_config_achse.ui16_ethercat_adr;
		END_IF

		(*-----------------------Weiterschaltbedingungen----------------------------*)
		fb_state_entry.i16_next_step := 7;

(*=======================================================*)
	7:	(* Spezifische NC-Achsparameter auslesen *)
		IF fb_state_entry.E THEN
			fb_axis.i16_nc_parameter_nummer := AxisMinSoftPosLimit;
			st_drive_cmd.enu_cmd := READ_NC_PARAMETER;
		END_IF

		(*-----------------------Weiterschaltbedingungen----------------------------*)
		IF st_drive_cmd.enu_cmd = NO_COMMAND THEN
			lr_MinSoftPosLimit := fb_axis.r_wert_nc_read_parameter;
			fb_state_entry.i16_next_step := 8;
		END_IF


(*=======================================================*)
	8:	(* Spezifische NC-Achsparameter auslesen *)
		IF fb_state_entry.E THEN
			fb_axis.i16_nc_parameter_nummer := AxisMaxSoftPosLimit;
			st_drive_cmd.enu_cmd := READ_NC_PARAMETER;
		END_IF

		(*-----------------------Weiterschaltbedingungen----------------------------*)
		IF st_drive_cmd.enu_cmd = NO_COMMAND THEN
			lr_MaxSoftPosLimit := fb_axis.r_wert_nc_read_parameter;
			fb_state_entry.i16_next_step := FEHLER; (*in Fehler gehen damit die Achsen resetet werden. Sonst steigen die Achsen bei einem TC Restart aus*)
		END_IF

(*=======================================================*)
	INIT:
		IF fb_state_entry.E THEN
			fb_ton_wz.IN := FALSE;
			fb_ton_uez.IN	:= FALSE;
			fb_ton_quitt.IN := FALSE;
			(* Reset Stoermeldungen *)
			st_sm.b_achse_nicht_auf_startpos := FALSE;
			st_sm.b_achsfehler := FALSE;
			st_sm.b_devicefehler := FALSE;
			st_sm.b_keine_verfahrfreigabe := FALSE;
			st_sm.b_ende_skalierungs_nocke := FALSE;
			st_sm.b_ende_camming_nocke := FALSE;
			st_sm.b_skalierung_noch_aktiv := FALSE;
			b_start_in:=FALSE;
			st_ctrl_out.b_busy:=FALSE;
			st_ctrl_out.b_fehler := FALSE;
			st_ctrl_out.b_fertig := FALSE;

			st_ctrl_out.b_bereit := FALSE;
			st_ctrl_out.b_prebereit := FALSE;
			sm_kein_nocken_definiert := FALSE;

			fb_axis.lr_soll_geschwindigkeit := gst_datensatz.st_wkz.r_auto_y;

			st_geschwindigkeiten.lr_verzoegerung := lr_decceleration_normal;
		END_IF

		(*-----------------------Weiterschaltbedingungen----------------------------*)
		IF st_ctrl_in.b_preinit THEN
			fb_state_entry.i16_next_step := 15;
		END_IF

(*=======================================================*)
	15:	(* Reglerfreigabe wegnehmen *)
		IF fb_state_entry.E THEN
			st_drive_cmd.enu_cmd := POWER_DISABLE;
		END_IF

		(*-----------------------Weiterschaltbedingungen----------------------------*)
		IF st_drive_cmd.enu_cmd = NO_COMMAND THEN
			fb_state_entry.i16_next_step := 20;
		END_IF

(*=======================================================*)
	20:	(* Überprüfe Nullpunktverschiebung des Absolutwertgebers auf Korrektheit *)
		IF fb_state_entry.E THEN
			fb_axis.i16_nc_parameter_nummer := AxisEncoderOffset;	(* vom Datentyp MC_AxisParameter *)
			st_drive_cmd.enu_cmd := READ_NC_PARAMETER;
		END_IF

		(*-----------------------Weiterschaltbedingungen----------------------------*)
		IF st_drive_cmd.enu_cmd = NO_COMMAND THEN
			IF fb_axis.r_wert_nc_read_parameter = gst_datensatz.st_md.st_md_y_achse.lr_nullpunktverschiebung THEN
				fb_state_entry.i16_next_step := 35;	(* Reglerfreigabe setzen *)
			ELSE
				fb_state_entry.i16_next_step := 25;	(* Nullpunktverschiebung schreiben *)
			END_IF
		END_IF

(*=======================================================*)
	25:	(* Nullpunktverschiebung hat sich geändert, deshalb erst Null reinschreiben, um keinen Additionsfehler zu machen, *)
		(* weil der Wert der Verschiebung beim Neustart komplett auf die Achse geschrieben wird *)
		IF fb_state_entry.E THEN
			fb_axis.i16_nc_parameter_nummer := AxisEncoderOffset;
			fb_axis.r_wert_nc_write_parameter := 0.0;
			st_drive_cmd.enu_cmd := WRITE_NC_PARAMETER;
		END_IF

		(*-----------------------Weiterschaltbedingungen----------------------------*)
		IF st_drive_cmd.enu_cmd = NO_COMMAND THEN
			fb_state_entry.i16_next_step := 30;
		END_IF

(*=======================================================*)
	30:	(* Aktuelle Nullpunktverschiebung des Absolutwertgebers an die Achse senden *)
		IF fb_state_entry.E THEN
			fb_axis.i16_nc_parameter_nummer := AxisEncoderOffset;
			fb_axis.r_wert_nc_write_parameter := gst_datensatz.st_md.st_md_y_achse.lr_nullpunktverschiebung;
			st_drive_cmd.enu_cmd := WRITE_NC_PARAMETER;
		END_IF

		(*-----------------------Weiterschaltbedingungen----------------------------*)
		IF st_drive_cmd.enu_cmd = NO_COMMAND THEN
			fb_state_entry.i16_next_step := 35;
		END_IF

(*=======================================================*)
	35:	(* Reglerfreigabe setzen , Reset wird bei Bedarf automatisch ausgeführt*)
		IF fb_state_entry.E THEN
			st_drive_cmd.enu_cmd := POWER_ENABLE;
		END_IF

		(*-----------------------Weiterschaltbedingungen----------------------------*)
		IF st_drive_cmd.enu_cmd = NO_COMMAND THEN
			fb_state_entry.i16_next_step := 40;
		END_IF

(*=======================================================*)
	40:	(* Nullpunktverschiebung ist geschrieben *)
		IF fb_state_entry.E THEN
			st_ctrl_out.b_prebereit := TRUE;
		END_IF

		(*-----------------------Weiterschaltbedingungen----------------------------*)
		IF st_ctrl_in.b_init THEN
			fb_state_entry.i16_next_step := 45;
		END_IF

(*=======================================================*)
	45: (* Warte auf Startsignal zum Positionieren *)

		(*-----------------------Weiterschaltbedingungen----------------------------*)
		IF st_ctrl_in.b_start THEN
			fb_state_entry.i16_next_step := 50;
		END_IF

(*=======================================================*)
	50: (* Positioniere Achse auf ausgelesene Slaveposition *)
		IF fb_state_entry.E THEN
			fb_axis.st_position.r_soll := ST_Z_Achse.lr_slave_position;
			st_drive_cmd.enu_cmd := MOVE_ABSOLUTE;
		END_IF

		(*-----------------------Weiterschaltbedingungen----------------------------*)
		IF st_drive_cmd.enu_cmd = NO_COMMAND THEN
			fb_state_entry.i16_next_step := 60;
		END_IF

(*=======================================================*)
	60: (* Warte bis Y-Achse gekoppelt wurde *)
		IF fb_state_entry.E THEN
			st_ctrl_out.b_fertig := TRUE;
		END_IF

		(*-----------------------Weiterschaltbedingungen----------------------------*)
		IF y_achse.NcToPlc.CoupleState = 3 THEN
			st_ctrl_out.b_fertig := FALSE;
			fb_state_entry.i16_next_step := BEREIT;
		END_IF

(*=======================================================*)
	BEREIT:
		IF fb_state_entry.E THEN
			st_ctrl_out.b_bereit := TRUE;
			enu_cmd_in:=NO_COMMAND;
		END_IF

		(*-----------------------Weiterschaltbedingungen----------------------------*)
		IF fb_r_trig_start.Q THEN
			st_ctrl_out.b_fertig_2 := FALSE;
			fb_state_entry.i16_next_step := 110;
		END_IF

		IF 	fb_r_trig_start_in.Q THEN		(*neu! zum Starten einer Positionierung von einem externen Prg.*)
			st_ctrl_out.b_fertig := FALSE;
			fb_state_entry.i16_next_step := 102;
		END_IF

		IF fb_state_entry.X THEN
			st_ctrl_out.b_fertig := FALSE;
			st_ctrl_out.b_busy:=TRUE;
		END_IF

(*=======================================================*)
	102:
		IF 	fb_state_entry.E THEN
			b_start_in:=FALSE;
		END_IF

		(*-----------------------Weiterschaltbedingungen----------------------------*)
		IF 	st_drive_cmd.enu_cmd = NO_COMMAND THEN
			fb_state_entry.i16_next_step := 104;
		END_IF

(*=======================================================*)
	104: (* Positioniere Achse  *)
		IF 	fb_state_entry.E THEN
			fb_axis.st_position.r_soll := lr_Achspos_in ;
			fb_axis.lr_soll_geschwindigkeit:=lr_Velo_in;
			st_drive_cmd.enu_cmd := enu_cmd_in;
		END_IF

		(*-----------------------Weiterschaltbedingungen----------------------------*)
		IF 	st_drive_cmd.enu_cmd = NO_COMMAND THEN
			st_ctrl_out.b_fertig := TRUE;
			fb_state_entry.i16_next_step := BEREIT;
		END_IF

		IF 	fb_state_entry.X THEN
			st_ctrl_out.b_busy:=FALSE;
		END_IF

(*=======================================================*)
	110: (* Fallunterscheidung *)
		CASE gst_datensatz.st_md.i16_typ_zelle OF
			KEINE_ZELLE:
				;

			BESTUECKZELLE_1700:
				(*-----------------------Weiterschaltbedingungen----------------------------*)
				fb_state_entry.i16_next_step := 200;

			RASTERFOLIE:
				(*-----------------------Weiterschaltbedingungen----------------------------*)
				fb_state_entry.i16_next_step := 120;

		END_CASE

(*=======================================================*)
	120: (* Positioniere Achse auf  0-Koordinate  des ISK *)
		IF fb_state_entry.E THEN
			fb_axis.st_position.r_soll := 	gst_datensatz.st_isk.lr_pos_y_0 +
										gst_datensatz.st_wkz.lr_offset_y_pos_0 +
										gst_datensatz.st_wt.lr_offset_y_pos_0 +
										gst_datensatz.st_md.lr_offset_y_pos_0 +
										gst_datensatz.st_bestueckprogramm.lr_y[0];
			st_drive_cmd.enu_cmd := MOVE_ABSOLUTE;
		END_IF

		(*-----------------------Weiterschaltbedingungen----------------------------*)
		IF st_drive_cmd.enu_cmd = NO_COMMAND THEN
			st_ctrl_out.b_fertig := TRUE;
			st_ctrl_out.b_busy:=FALSE;
			fb_state_entry.i16_next_step := 300;
		END_IF

(*=======================================================*)
	200:
		IF fb_state_entry.E THEN
			st_ctrl_out.b_fertig := TRUE;
			st_ctrl_out.b_busy:=FALSE;
		END_IF

		(*-----------------------Weiterschaltbedingungen----------------------------*)
		IF st_ctrl_in.b_start_2 THEN
			st_ctrl_out.b_fertig := FALSE;
			fb_state_entry.i16_next_step := 210;
		END_IF

(*=======================================================*)
	210: (* Positioniere Achse auf gewünschte Position *)
		IF fb_state_entry.E THEN
			fb_axis.st_position.r_soll :=  ST_Z_Achse.lr_slave_position;
			st_drive_cmd.enu_cmd := MOVE_ABSOLUTE;
		END_IF

		(*-----------------------Weiterschaltbedingungen----------------------------*)
		IF st_drive_cmd.enu_cmd = NO_COMMAND THEN
			fb_state_entry.i16_next_step := 220;
		END_IF

(*=======================================================*)
	220: (* Warte bis Y-Achse gekoppelt wurde *)
		IF fb_state_entry.E THEN
			st_ctrl_out.b_fertig_2 := TRUE;
		END_IF

		(*-----------------------Weiterschaltbedingungen----------------------------*)
		IF y_achse.NcToPlc.CoupleState = 3 THEN
			st_ctrl_out.b_fertig_2 := FALSE;
			fb_state_entry.i16_next_step := BEREIT;
		END_IF

(*=======================================================*)
	300:(* Verfahre Y-Achse undwarte auf Start von Z-Achse *)

		(*-----------------------Weiterschaltbedingungen----------------------------*)
		(* Verfahre Y-Achse *)
		IF	gst_datensatz.st_md.i16_typ_zelle = RASTERFOLIE AND
			ST_Rasterfolienmontage.b_start_y_Achse THEN
			fb_state_entry.i16_next_step := 310;
		END_IF

		(* Warte auf Start von Z-Achse *)
		IF st_ctrl_in.b_start_2 THEN
			st_ctrl_out.b_fertig := FALSE;
			fb_state_entry.i16_next_step := 350;
		END_IF

(*=======================================================*)
	310: (* Positioniere Achse  *)
		IF fb_state_entry.E THEN
			fb_axis.st_position.r_soll := 	lr_tmp_Achspos;
			st_drive_cmd.enu_cmd := MOVE_ABSOLUTE;
		END_IF

		(*-----------------------Weiterschaltbedingungen----------------------------*)
		IF st_drive_cmd.enu_cmd = NO_COMMAND THEN
			fb_state_entry.i16_next_step := 300;
			ST_Rasterfolienmontage.b_start_y_Achse:=FALSE;
		END_IF


(*=======================================================*)
	350: (* Positioniere Achse auf gewünschte Position am Ende der Kurvenscheibe *)
		IF fb_state_entry.E THEN
			fb_axis.st_position.r_soll :=  ST_Z_Achse.lr_slave_position;
			st_drive_cmd.enu_cmd := MOVE_ABSOLUTE;
		END_IF

		(*-----------------------Weiterschaltbedingungen----------------------------*)
		IF st_drive_cmd.enu_cmd = NO_COMMAND THEN
			fb_state_entry.i16_next_step := 360;
		END_IF

(*=======================================================*)
	360: (* Warte bis Y-Achse gekoppelt wurde *)
		IF fb_state_entry.E THEN
			st_ctrl_out.b_fertig_2 := TRUE;
		END_IF

		(*-----------------------Weiterschaltbedingungen----------------------------*)
		IF y_achse.NcToPlc.CoupleState = 3 THEN
			st_ctrl_out.b_fertig_2 := FALSE;
			fb_state_entry.i16_next_step := BEREIT;
		END_IF

(*=======================================================*)
	FEHLER:
		IF fb_state_entry.E THEN
			st_ctrl_out.b_fehler := TRUE;
			fb_ton_quitt.IN := FALSE;
			st_ctrl_out.b_busy:=FALSE;
		END_IF

		IF st_ctrl_in.b_stop AND NOT y_achse.Status.HasBeenStopped THEN
			st_drive_cmd.enu_cmd := STOP_AXIS;
		END_IF

		IF st_ctrl_in.b_halt AND y_achse.Status.Moving THEN
			st_drive_cmd.enu_cmd := HALT_AXIS;
			st_geschwindigkeiten.lr_verzoegerung := lr_decceleration_nothalt;
		END_IF

		(*-----------------------Weiterschaltbedingungen----------------------------*)
		IF st_ctrl_in.b_quitt AND NOT fb_state_entry.E THEN
			st_ctrl_out.b_fehler := FALSE;
			st_drive_cmd.enu_cmd := RESET;
			fb_ton_quitt.IN := TRUE;
		END_IF

		IF fb_ton_quitt.Q THEN
			fb_ton_quitt.IN := FALSE;
			fb_state_entry.i16_next_step := INIT;
		END_IF

(*=======================================================*)
	STOP:
		IF fb_state_entry.E THEN
			st_ctrl_out.b_busy:=FALSE;
			IF y_achse.NcToPlc.CoupleState = 0 THEN
				st_drive_cmd.enu_cmd := STOP_AXIS;
			END_IF
		END_IF

		(*-----------------------Weiterschaltbedingungen----------------------------*)
		IF st_drive_cmd.enu_cmd = NO_COMMAND AND y_achse.Status.NotMoving THEN
			fb_state_entry.i16_next_step := STILLSTAND;
		END_IF

(*=======================================================*)
	STILLSTAND:
		IF fb_state_entry.E THEN
			st_drive_cmd.enu_cmd := POWER_DISABLE;
			fb_ton_quitt.IN := FALSE;
		END_IF

		(*-----------------------Weiterschaltbedingungen----------------------------*)
		IF st_ctrl_in.b_quitt AND NOT fb_state_entry.E THEN
			fb_ton_quitt.IN := TRUE;
		END_IF

		IF fb_ton_quitt.Q THEN
			fb_ton_quitt.IN := FALSE;
			fb_state_entry.i16_next_step := INIT;
		END_IF

(*=======================================================*)
	HALT:
		IF fb_state_entry.E THEN
			IF y_achse.NcToPlc.CoupleState = 0 THEN
				st_drive_cmd.enu_cmd := HALT_AXIS;
				st_geschwindigkeiten.lr_verzoegerung := lr_decceleration_nothalt;
			END_IF
			fb_ton_quitt.IN := FALSE;
		END_IF

		(*-----------------------Weiterschaltbedingungen----------------------------*)
		IF st_ctrl_in.b_quitt AND NOT fb_state_entry.E THEN
			fb_ton_quitt.IN := TRUE;
		END_IF

		IF fb_ton_quitt.Q THEN
			fb_ton_quitt.IN := FALSE;
			fb_state_entry.i16_next_step := INIT;
		END_IF

(*=======================================================*)
	HANDRAD:	(* Überprüfe Nullpunktverschiebung des Absolutwertgebers auf Korrektheit *)
		IF fb_state_entry.E THEN
			st_ctrl_out.b_fehler := TRUE;
			fb_axis.i16_nc_parameter_nummer := AxisEncoderOffset;
			st_drive_cmd.enu_cmd := READ_NC_PARAMETER;
		END_IF

		(*-----------------------Weiterschaltbedingungen----------------------------*)
		IF st_drive_cmd.enu_cmd = NO_COMMAND THEN
			IF fb_axis.r_wert_nc_read_parameter = gst_datensatz.st_md.st_md_y_achse.lr_nullpunktverschiebung THEN
				fb_state_entry.i16_next_step := 2040;	(* Jogbetrieb *)
			ELSE
				fb_state_entry.i16_next_step := 2010;	(* Reglerfreigabe nehmen und Nullpunktverschiebung schreiben *)
			END_IF
		END_IF

(*=======================================================*)
	2010:	(* Reglerfreigabe wegnehmen , damit Nullpunktverschiebung geschrieben werden kannt*)
		IF fb_state_entry.E THEN
			st_drive_cmd.enu_cmd := POWER_DISABLE;
		END_IF

		(*-----------------------Weiterschaltbedingungen----------------------------*)
		IF st_drive_cmd.enu_cmd = NO_COMMAND THEN
			fb_state_entry.i16_next_step := 2020;
		END_IF

(*=======================================================*)
	2020:	(* Nullpunktverschiebung hat sich geändert, deshalb erst Null reinschreiben, um keinen Additionsfehler zu machen, *)
			(* weil der Wert der Verschiebung beim Neustart komplett auf die Achse geschrieben wird *)
		IF fb_state_entry.E THEN
			fb_axis.i16_nc_parameter_nummer := AxisEncoderOffset;
			fb_axis.r_wert_nc_write_parameter := 0.0;
			st_drive_cmd.enu_cmd := WRITE_NC_PARAMETER;
		END_IF

		(*-----------------------Weiterschaltbedingungen----------------------------*)
		IF st_drive_cmd.enu_cmd = NO_COMMAND THEN
			fb_state_entry.i16_next_step := 2030;
		END_IF

(*=======================================================*)
	2030:	(* Aktuelle Nullpunktverschiebung des Absolutwertgebers an die Achse senden *)
		IF fb_state_entry.E THEN
			fb_axis.i16_nc_parameter_nummer := AxisEncoderOffset;
			fb_axis.r_wert_nc_write_parameter := gst_datensatz.st_md.st_md_y_achse.lr_nullpunktverschiebung;
			st_drive_cmd.enu_cmd := WRITE_NC_PARAMETER;
		END_IF

		(*-----------------------Weiterschaltbedingungen----------------------------*)
		IF st_drive_cmd.enu_cmd = NO_COMMAND THEN
			fb_state_entry.i16_next_step := 2040;
		END_IF

(*=======================================================*)
	2040:	(* Jogbetrieb *)
		IF fb_state_entry.E THEN
			fb_axis.lr_soll_geschwindigkeit := st_geschwindigkeiten.lr_jog;
		END_IF

		IF ST_Euchner_Handbedienpult.i16_Handrad_delta > 0 THEN
			st_drive_cmd.enu_cmd := JOG_VORWAERTS;
		ELSIF ST_Euchner_Handbedienpult.i16_Handrad_delta < 0 THEN
			st_drive_cmd.enu_cmd := JOG_RUECKWAERTS;
		ELSIF  y_achse.Status.Moving THEN
			st_drive_cmd.enu_cmd := JOG_STOP;
		END_IF

		IF fb_r_trig_taste_plus.Q THEN
			fb_state_entry.i16_next_step := MOTORBREMSE_AUF;
		END_IF
		IF fb_r_trig_taste_minus.Q THEN
			fb_state_entry.i16_next_step := MOTORBREMSE_ZU;
		END_IF

		(*-----------------------Weiterschaltbedingungen----------------------------*)
		IF gi16_betriebsart <> HAND OR NOT b_hand_dialog_aktiv THEN
			fb_state_entry.i16_next_step := 2050;
		END_IF

(*=======================================================*)
	2050:
		IF fb_state_entry.E THEN
			st_drive_cmd.enu_cmd := ABORT;
		END_IF

		(*-----------------------Weiterschaltbedingungen----------------------------*)
		IF st_drive_cmd.enu_cmd = NO_COMMAND THEN
			fb_state_entry.i16_next_step := 2060;
		END_IF

(*=======================================================*)
	2060:
		IF fb_state_entry.E THEN
			fb_axis.w_idn := P_0_IDN + 96;
			fb_axis.ui16_soeparam_write_value := 0;	(* Motorbremse im Automatikbetrieb für reguläres Fahren *)
			st_drive_cmd.enu_cmd := SOE_WRITE_PARAM;
		END_IF

		(*-----------------------Weiterschaltbedingungen----------------------------*)
		IF st_drive_cmd.enu_cmd = NO_COMMAND THEN
			fb_state_entry.i16_next_step := 2070;
		END_IF

(*=======================================================*)
	2070:	(* Reglerfreigabe wegnehmen *)
		IF fb_state_entry.E THEN
			st_drive_cmd.enu_cmd := POWER_DISABLE;
		END_IF

		(*-----------------------Weiterschaltbedingungen----------------------------*)
		IF st_drive_cmd.enu_cmd = NO_COMMAND THEN
			st_ctrl_out.b_fehler := FALSE;
			fb_state_entry.i16_next_step := INIT;
		END_IF

(*=======================================================*)
	MOTORBREMSE_AUF:
		IF fb_state_entry.E THEN
			st_drive_cmd.enu_cmd := ABORT;
		END_IF

		(*-----------------------Weiterschaltbedingungen----------------------------*)
		IF st_drive_cmd.enu_cmd = NO_COMMAND THEN
			fb_state_entry.i16_next_step := 2110;
		END_IF

(*=======================================================*)
	2110:	(* Reglerfreigabe wegnehmen *)
		IF fb_state_entry.E THEN
			st_drive_cmd.enu_cmd := POWER_DISABLE;
		END_IF

		(*-----------------------Weiterschaltbedingungen----------------------------*)
		IF st_drive_cmd.enu_cmd = NO_COMMAND THEN
			fb_state_entry.i16_next_step := 2120;
		END_IF

(*=======================================================*)
	2120:	(* Bremse auf machen *)
		IF fb_state_entry.E THEN
			fb_axis.w_idn := P_0_IDN + 96;
			fb_axis.ui16_soeparam_write_value := 2;
			st_drive_cmd.enu_cmd := SOE_WRITE_PARAM;
		END_IF

		(*-----------------------Weiterschaltbedingungen----------------------------*)
		IF 	st_drive_cmd.enu_cmd = NO_COMMAND AND
			(gi16_betriebsart <> HAND OR
			NOT b_hand_dialog_aktiv OR
			ST_Euchner_Handbedienpult.i16_Handrad_delta > 0)
			THEN
				fb_state_entry.i16_next_step := HANDRAD;
		ELSIF fb_r_trig_taste_minus.Q THEN
			fb_state_entry.i16_next_step := MOTORBREMSE_ZU;
		END_IF

(*=======================================================*)
	MOTORBREMSE_ZU:
		IF fb_state_entry.E THEN
			st_drive_cmd.enu_cmd := ABORT;
		END_IF

		(*-----------------------Weiterschaltbedingungen----------------------------*)
		IF st_drive_cmd.enu_cmd = NO_COMMAND THEN
			fb_state_entry.i16_next_step := 2210;
		END_IF

(*=======================================================*)
	2210:	(* Reglerfreigabe setzen *)
		IF fb_state_entry.E THEN
			st_drive_cmd.enu_cmd := POWER_ENABLE;
		END_IF

		(*-----------------------Weiterschaltbedingungen----------------------------*)
		IF st_drive_cmd.enu_cmd = NO_COMMAND THEN
			fb_state_entry.i16_next_step := 2220;
		END_IF

(*=======================================================*)
	2220:	(* Bremse zu machen *)
		IF fb_state_entry.E THEN
			fb_axis.w_idn := P_0_IDN + 96;
			fb_axis.ui16_soeparam_write_value := 0;
			st_drive_cmd.enu_cmd := SOE_WRITE_PARAM;
		END_IF

		(*-----------------------Weiterschaltbedingungen----------------------------*)
		IF 	st_drive_cmd.enu_cmd = NO_COMMAND AND
			(gi16_betriebsart <> HAND OR
			NOT b_hand_dialog_aktiv OR
			ST_Euchner_Handbedienpult.i16_Handrad_delta > 0)
			THEN
				fb_state_entry.i16_next_step := HANDRAD;
		ELSIF fb_r_trig_taste_plus.Q THEN
			fb_state_entry.i16_next_step := MOTORBREMSE_AUF;
		END_IF

(*=======================================================*)
	NULLPUNKT_SETZEN:
		(* Aktuellen Jog beenden, sonst Probleme beim Softwareendschalter*)
		IF fb_state_entry.E THEN
			st_drive_cmd.enu_cmd := JOG_STOP;
		END_IF

		(*-----------------------Weiterschaltbedingungen----------------------------*)
		IF st_drive_cmd.enu_cmd = NO_COMMAND THEN
			fb_state_entry.i16_next_step := 2505;
		END_IF

(*=======================================================*)
	2505:
		(* 	Lese aktuelle Nullpunkt verschiebung von der Hardware. Der Benutze könnte einen falschen
			Wert eingetragen haben *)
		IF fb_state_entry.E THEN
			fb_axis.i16_nc_parameter_nummer := AxisEncoderOffset;
			st_drive_cmd.enu_cmd := READ_NC_PARAMETER;
		END_IF

		(*-----------------------Weiterschaltbedingungen----------------------------*)
		IF st_drive_cmd.enu_cmd = NO_COMMAND THEN
			gst_datensatz.st_md.st_md_y_achse.lr_nullpunktverschiebung := fb_axis.r_wert_nc_read_parameter;
			fb_state_entry.i16_next_step := 2510;
		END_IF

(*=======================================================*)
	2510:	(* Nullpunktverschiebung berechnen *)
		IF fb_state_entry.E THEN
			lr_pos_ohneverschiebung := axis_y_achse.st_visu.lr_position_ist - gst_datensatz.st_md.st_md_y_achse.lr_nullpunktverschiebung;

			gst_datensatz.st_md.st_md_y_achse.lr_nullpunktverschiebung := - lr_pos_ohneverschiebung;
		END_IF

		(*-----------------------Weiterschaltbedingungen----------------------------*)
		(* Aktiviere den wert in die Hardware *)
		fb_state_entry.i16_next_step := HANDRAD;

(*=======================================================*)
	INBETRIEBNAHME:	(* Überprüfe Nullpunktverschiebung des Absolutwertgebers auf Korrektheit *)
		IF fb_state_entry.E THEN
			fb_axis.i16_nc_parameter_nummer := AxisEncoderOffset;
			st_drive_cmd.enu_cmd := READ_NC_PARAMETER;
		END_IF

		(*-----------------------Weiterschaltbedingungen----------------------------*)
		IF st_drive_cmd.enu_cmd = NO_COMMAND THEN
			IF fb_axis.r_wert_nc_read_parameter = gst_datensatz.st_md.st_md_y_achse.lr_nullpunktverschiebung THEN
				fb_state_entry.i16_next_step := 5100;	(* Reversiersequenz*)
			ELSE
				fb_state_entry.i16_next_step := 5010;	(* Reglerfreigabe nehmen und Nullpunktverschiebung schreiben *)
			END_IF
		END_IF

(*=======================================================*)
	5010:	(* Reglerfreigabe wegnehmen, damit Nullpunktverschiebung geschrieben werden kannt*)
		IF fb_state_entry.E THEN
			st_drive_cmd.enu_cmd := POWER_DISABLE;
		END_IF

		(*-----------------------Weiterschaltbedingungen----------------------------*)
		IF st_drive_cmd.enu_cmd = NO_COMMAND THEN
			fb_state_entry.i16_next_step := 5020;
		END_IF

(*=======================================================*)
	5020:	(* Nullpunktverschiebung hat sich geändert, deshalb erst Null reinschreiben, um keinen Additionsfehler zu machen, *)
			(* weil der Wert der Verschiebung beim Neustart komplett auf die Achse geschrieben wird *)
		IF fb_state_entry.E THEN
			fb_axis.i16_nc_parameter_nummer := AxisEncoderOffset;
			fb_axis.r_wert_nc_write_parameter := 0.0;
			st_drive_cmd.enu_cmd := WRITE_NC_PARAMETER;
		END_IF

		(*-----------------------Weiterschaltbedingungen----------------------------*)
		IF st_drive_cmd.enu_cmd = NO_COMMAND THEN
			fb_state_entry.i16_next_step := 5030;
		END_IF

